# B&R Automation Studio project NAINV104C00R8L515F00 (part 14)

#### Act_OptP1023USSel.st
```iecst
ACTION Act_OptP1023USSel:

	IF tyP1023McSetHComm.tyUSSel.tyBtnSMEMA.bRtCompl = TRUE THEN
		tyP1023McSetHComm.tyUSSel.tyBtnSMEMA.bRtCompl	:= FALSE;

		tyP1023McSetHComm.tyUSSel.tyBtnSMEMA.bValue		:= TRUE;
		tyP1023McSetHComm.tyUSSel.tyBtnSMEMA.bRtLk		:= TRUE;

		tyP1023McSetHComm.tyUSSel.tyBtnHermes.bValue	:= FALSE;
		tyP1023McSetHComm.tyUSSel.tyBtnHermes.bRtLk		:= FALSE;

	ELSIF tyP1023McSetHComm.tyUSSel2.tyBtnSMEMA.bRtCompl = TRUE THEN
		tyP1023McSetHComm.tyUSSel2.tyBtnSMEMA.bRtCompl	:= FALSE;

		tyP1023McSetHComm.tyUSSel2.tyBtnSMEMA.bValue	:= TRUE;
		tyP1023McSetHComm.tyUSSel2.tyBtnSMEMA.bRtLk		:= TRUE;

		tyP1023McSetHComm.tyUSSel2.tyBtnHermes.bValue	:= FALSE;
		tyP1023McSetHComm.tyUSSel2.tyBtnHermes.bRtLk	:= FALSE;

	ELSIF tyP1023McSetHComm.tyUSSel.tyBtnHermes.bRtCompl = TRUE THEN
		tyP1023McSetHComm.tyUSSel.tyBtnHermes.bRtCompl	:= FALSE;

		tyP1023McSetHComm.tyUSSel.tyBtnSMEMA.bValue		:= FALSE;
		tyP1023McSetHComm.tyUSSel.tyBtnSMEMA.bRtLk		:= FALSE;

		tyP1023McSetHComm.tyUSSel.tyBtnHermes.bValue	:= TRUE;
		tyP1023McSetHComm.tyUSSel.tyBtnHermes.bRtLk		:= TRUE;

	ELSIF tyP1023McSetHComm.tyUSSel2.tyBtnHermes.bRtCompl = TRUE THEN //Added
		tyP1023McSetHComm.tyUSSel2.tyBtnHermes.bRtCompl	:= FALSE;

		tyP1023McSetHComm.tyUSSel2.tyBtnSMEMA.bValue	:= FALSE;
		tyP1023McSetHComm.tyUSSel2.tyBtnSMEMA.bRtLk		:= FALSE;

		tyP1023McSetHComm.tyUSSel2.tyBtnHermes.bValue	:= TRUE;
		tyP1023McSetHComm.tyUSSel2.tyBtnHermes.bRtLk	:= TRUE;

	END_IF

	//Upstream Selection

	IF tyP1023McSetHComm.tyGen.tyDrpDnUSSel.bRtCompl THEN

		tyP1023McSetHComm.tyGen.tyDrpDnUSSel.bRtCompl:= FALSE;

		IF tyP1023McSetHComm.tyGen.tyDrpDnUSSel.usiValueIdx = 0 THEN

			p_tyP1023McSetHCommUSSel ACCESS ADR(tyP1023McSetHComm.tyUSSel);
			p_tyP1023McSetHCommUSSMEMA ACCESS ADR(tyP1023McSetHComm.tyUSSMEMA);
			p_tyP1023McSetHCommUSHermes ACCESS ADR(tyP1023McSetHComm.tyUSHermes);

			fUIInRtStatOff(ADR(tyP1023McSetHComm.tyUSSel.tyLyr.uiRtStat));
			fUIInRtStatHide(ADR(tyP1023McSetHComm.tyUSSel2.tyLyr.uiRtStat));

		ELSIF tyP1023McSetHComm.tyGen.tyDrpDnUSSel.usiValueIdx = 1 THEN

			p_tyP1023McSetHCommUSSel ACCESS ADR(tyP1023McSetHComm.tyUSSel2);
			p_tyP1023McSetHCommUSSMEMA ACCESS ADR(tyP1023McSetHComm.tyUSSMEMA2);
			p_tyP1023McSetHCommUSHermes ACCESS ADR(tyP1023McSetHComm.tyUSHermes2);

			fUIInRtStatOff(ADR(tyP1023McSetHComm.tyUSSel2.tyLyr.uiRtStat));
			fUIInRtStatHide(ADR(tyP1023McSetHComm.tyUSSel.tyLyr.uiRtStat));

		END_IF

	END_IF

END_ACTION
```

#### Act_OptP1023DSSel.st
```iecst
ACTION Act_OptP1023DSSel:

	IF tyP1023McSetHComm.tyDSSel.tyBtnSMEMA.bRtCompl = TRUE THEN
		tyP1023McSetHComm.tyDSSel.tyBtnSMEMA.bRtCompl	:= FALSE;

		tyP1023McSetHComm.tyDSSel.tyBtnSMEMA.bValue		:= TRUE;
		tyP1023McSetHComm.tyDSSel.tyBtnSMEMA.bRtLk		:= TRUE;

		tyP1023McSetHComm.tyDSSel.tyBtnHermes.bValue	:= FALSE;
		tyP1023McSetHComm.tyDSSel.tyBtnHermes.bRtLk		:= FALSE;

	ELSIF tyP1023McSetHComm.tyDSSel.tyBtnHermes.bRtCompl = TRUE THEN
		tyP1023McSetHComm.tyDSSel.tyBtnHermes.bRtCompl	:= FALSE;

		tyP1023McSetHComm.tyDSSel.tyBtnSMEMA.bValue		:= FALSE;
		tyP1023McSetHComm.tyDSSel.tyBtnSMEMA.bRtLk		:= FALSE;

		tyP1023McSetHComm.tyDSSel.tyBtnHermes.bValue	:= TRUE;
		tyP1023McSetHComm.tyDSSel.tyBtnHermes.bRtLk		:= TRUE;
	ELSIF tyP1023McSetHComm.tyDSSel2.tyBtnSMEMA.bRtCompl = TRUE THEN
		tyP1023McSetHComm.tyDSSel2.tyBtnSMEMA.bRtCompl	:= FALSE;

		tyP1023McSetHComm.tyDSSel2.tyBtnSMEMA.bValue		:= TRUE;
		tyP1023McSetHComm.tyDSSel2.tyBtnSMEMA.bRtLk		:= TRUE;

		tyP1023McSetHComm.tyDSSel2.tyBtnHermes.bValue	:= FALSE;
		tyP1023McSetHComm.tyDSSel2.tyBtnHermes.bRtLk		:= FALSE;

	ELSIF  tyP1023McSetHComm.tyDSSel2.tyBtnHermes.bRtCompl = TRUE THEN
		tyP1023McSetHComm.tyDSSel2.tyBtnHermes.bRtCompl	:= FALSE;

		tyP1023McSetHComm.tyDSSel2.tyBtnSMEMA.bValue		:= FALSE;
		tyP1023McSetHComm.tyDSSel2.tyBtnSMEMA.bRtLk		:= FALSE;

		tyP1023McSetHComm.tyDSSel2.tyBtnHermes.bValue	:= TRUE;
		tyP1023McSetHComm.tyDSSel2.tyBtnHermes.bRtLk		:= TRUE;

	END_IF

	//Dsstream Selection
	IF tyP1023McSetHComm.tyGen.tyDrpDnDSSel.bRtCompl THEN

		tyP1023McSetHComm.tyGen.tyDrpDnDSSel.bRtCompl:= FALSE;

		IF tyP1023McSetHComm.tyGen.tyDrpDnDSSel.usiValueIdx = 0 THEN

			p_tyP1023McSetHCommDSSel ACCESS ADR(tyP1023McSetHComm.tyDSSel);
			p_tyP1023McSetHCommDSSMEMA ACCESS ADR(tyP1023McSetHComm.tyDSSMEMA);
			p_tyP1023McSetHCommDSHermes ACCESS ADR(tyP1023McSetHComm.tyDSHermes);

			fUIInRtStatOff(ADR(tyP1023McSetHComm.tyDSSel.tyLyr.uiRtStat));
			fUIInRtStatHide(ADR(tyP1023McSetHComm.tyDSSel2.tyLyr.uiRtStat));

		ELSIF tyP1023McSetHComm.tyGen.tyDrpDnDSSel.usiValueIdx = 1 THEN

			p_tyP1023McSetHCommDSSel ACCESS ADR(tyP1023McSetHComm.tyDSSel2);
			p_tyP1023McSetHCommDSSMEMA ACCESS ADR(tyP1023McSetHComm.tyDSSMEMA2);
			p_tyP1023McSetHCommDSHermes ACCESS ADR(tyP1023McSetHComm.tyDSHermes2);

			fUIInRtStatOff(ADR(tyP1023McSetHComm.tyDSSel2.tyLyr.uiRtStat));
			fUIInRtStatHide(ADR(tyP1023McSetHComm.tyDSSel.tyLyr.uiRtStat));

		END_IF

	END_IF

END_ACTION
```

#### Act_OptP1023Keypad.st
```iecst
ACTION Act_OptP1023Keypad:

	IF fUIOutRtStatTPIsOpen(ADR(tyP1023McSetHComm.tyUSHermes.tyNumSndAliveTm.uiRtStat)) = TRUE THEN
		tyProperty.tyKeypad.tyTxtTitle.sTxt	:= tyP1023McSetHComm.tyUSHermes.tyNumSndAliveTm.sKeypadTitle;

	ELSIF fUIOutRtStatTPIsOpen(ADR(tyP1023McSetHComm.tyUSHermes.tyNumLaneID.uiRtStat)) = TRUE THEN
		tyProperty.tyKeypad.tyTxtTitle.sTxt	:= tyP1023McSetHComm.tyUSHermes.tyNumLaneID.sKeypadTitle;

	ELSIF fUIOutRtStatTPIsOpen(ADR(tyP1023McSetHComm.tyUSHermes.tyStringHostAddr.uiRtStat)) = TRUE THEN
		tyProperty.tyKeypad.tyTxtTitle.sTxt	:= tyP1023McSetHComm.tyUSHermes.tyStringHostAddr.sKeypadTitle;

	ELSIF fUIOutRtStatTPIsOpen(ADR(tyP1023McSetHComm.tyUSHermes.tyNumHostPort.uiRtStat)) = TRUE THEN
		tyProperty.tyKeypad.tyTxtTitle.sTxt	:= tyP1023McSetHComm.tyUSHermes.tyNumHostPort.sKeypadTitle;

	ELSIF fUIOutRtStatTPIsOpen(ADR(tyP1023McSetHComm.tyDSHermes.tyNumSndAliveTm.uiRtStat)) = TRUE THEN
		tyProperty.tyKeypad.tyTxtTitle.sTxt	:= tyP1023McSetHComm.tyDSHermes.tyNumSndAliveTm.sKeypadTitle;

	ELSIF fUIOutRtStatTPIsOpen(ADR(tyP1023McSetHComm.tyDSHermes.tyNumLaneID.uiRtStat)) = TRUE THEN
		tyProperty.tyKeypad.tyTxtTitle.sTxt	:= tyP1023McSetHComm.tyDSHermes.tyNumLaneID.sKeypadTitle;

	ELSIF fUIOutRtStatTPIsOpen(ADR(tyP1023McSetHComm.tyDSHermes.tyNumSvrPort.uiRtStat)) = TRUE THEN
		tyProperty.tyKeypad.tyTxtTitle.sTxt	:= tyP1023McSetHComm.tyDSHermes.tyNumSvrPort.sKeypadTitle;

	END_IF

END_ACTION
```

#### Act_EntP1024Disp.st
```iecst
ACTION Act_EntP1024Disp:

	//Access Address
	p_tyC0004Navi ACCESS ADR(tyP1024McSetAntiGap.tyNaviBack);

	p_tyC0005Main ACCESS ADR(tyCommon.tyMain);

	p_tyC0006Set ACCESS ADR(tyCommon.tySet);

	p_tyC0007Notif ACCESS ADR(tyCommon.tyNotif);

	p_tyC0008MsgBox ACCESS ADR(tyP1024McSetAntiGap.tyMsgBoxHide);

	p_tyC0009Info ACCESS ADR(tyCommon.tyInfo);

	p_tyC0011Loading ACCESS ADR(tyCommon.tyLoading);

	p_tyP1024McSetAntiGap ACCESS ADR(tyP1024McSetAntiGap.tyAntiGap);

	//Backup Param
	tyP1024McSetAntiGap.tyAntiGapBkUp	:= tyP1024McSetAntiGap.tyAntiGap;

END_ACTION
```

#### Act_ExitP1024.st
```iecst
ACTION Act_ExitP1024:

	IF tyCommon.tySet.tyBtnSave.uiMaskRtStat.0 = FALSE THEN
		usiChgPage	:= 1;

	ELSE

		p_tyC0008MsgBox ACCESS ADR(tyP1024McSetAntiGap.tyMsgBoxExitAsk);

		IF tyP1024McSetAntiGap.tyMsgBoxExitAsk.tyBtnYes.bRtCompl = TRUE THEN
			tyP1024McSetAntiGap.tyMsgBoxExitAsk.tyBtnYes.bRtCompl	:= FALSE;
			tyP1024McSetAntiGap.tyMsgBoxExitAsk.tyBtnYes.bValue		:= FALSE;

			p_tyC0008MsgBox ACCESS ADR(tyP1024McSetAntiGap.tyMsgBoxHide);

			//Restore Param
			tyP1024McSetAntiGap.tyAntiGap	:= tyP1024McSetAntiGap.tyAntiGapBkUp;

			fUIInRtStatOff(ADR(tyCommon.tySet.tyBtnSave.uiMaskRtStat));

			usiChgPage	:= 1;

		ELSIF tyP1024McSetAntiGap.tyMsgBoxExitAsk.tyBtnNo.bRtCompl = TRUE THEN
			tyP1024McSetAntiGap.tyMsgBoxExitAsk.tyBtnNo.bRtCompl	:= FALSE;
			tyP1024McSetAntiGap.tyMsgBoxExitAsk.tyBtnNo.bValue		:= FALSE;

			p_tyC0008MsgBox ACCESS ADR(tyP1024McSetAntiGap.tyMsgBoxHide);

			eChgPage	:= eCurrPage;
			usiChgPage	:= 0;

		END_IF

	END_IF

END_ACTION
```

#### Act_OptP1024Navi.st
```iecst
ACTION Act_OptP1024Navi:

	IF tyP1024McSetAntiGap.tyNaviBack.tyBtnBack.bRtCompl = TRUE THEN
		tyP1024McSetAntiGap.tyNaviBack.tyBtnBack.bRtCompl	:= FALSE;

		eChgPage	:= UIP1020McSetNavi;

	END_IF

END_ACTION
```

#### Act_OptP1024Save.st
```iecst
ACTION Act_OptP1024Save:

	IF 	tyP1024McSetAntiGap.tyAntiGap.tyNumLftSenOff.bRtCompl OR tyP1024McSetAntiGap.tyAntiGap.tyNumRgtSenOff.bRtCompl THEN

		fUIInRtStatHide(ADR(tyCommon.tySet.tyBtnSave.uiMaskRtStat));

		tyP1024McSetAntiGap.tyAntiGap.tyNumLftSenOff.bRtCompl	:= FALSE;
		tyP1024McSetAntiGap.tyAntiGap.tyNumRgtSenOff.bRtCompl	:= FALSE;

	END_IF

	IF tyCommon.tySet.tyBtnSave.bRtCompl = TRUE THEN
		//Save Param
		tyMcParamWr.tyConvLftSenAntiGapDly.diSigOffTm	:= tyP1024McSetAntiGap.tyAntiGap.tyNumLftSenOff.diValue;
		tyMcParamWr.tyConvRgtSenAntiGapDly.diSigOffTm	:= tyP1024McSetAntiGap.tyAntiGap.tyNumRgtSenOff.diValue;

		eMcParamAct	:= McParamActWrite;

		IF p_eMcParamStat = McParamActWrite AND p_eMcParamStatus = Done THEN
			eMcParamAct	:= McParamActIdle;

			//Backup Param
			tyP1024McSetAntiGap.tyAntiGapBkUp	:= tyP1024McSetAntiGap.tyAntiGap;

			tyCommon.tySet.tyBtnSave.bRtCompl	:= FALSE;

			fUIInRtStatOff(ADR(tyCommon.tySet.tyBtnSave.uiMaskRtStat));

		ELSIF p_eMcParamStatus = Error THEN
			p_tyC0008MsgBox ACCESS ADR(tyP1024McSetAntiGap.tyMsgBoxSaveErr);

			IF tyP1021McSetGen.tyMsgBoxSaveErr.tyBtnNo.bRtCompl = TRUE THEN
				tyP1021McSetGen.tyMsgBoxSaveErr.tyBtnNo.bRtCompl	:= FALSE;
				tyP1021McSetGen.tyMsgBoxSaveErr.tyBtnNo.bValue		:= FALSE;

				p_tyC0008MsgBox ACCESS ADR(tyP1024McSetAntiGap.tyMsgBoxHide);

				//Restore Param
				tyP1024McSetAntiGap.tyAntiGap	:= tyP1024McSetAntiGap.tyAntiGapBkUp;
				tyMcParamWr						:= p_tyMcParamCurr;

				tyCommon.tySet.tyBtnSave.bRtCompl	:= FALSE;

				fUIInRtStatOff(ADR(tyCommon.tySet.tyBtnSave.uiMaskRtStat));

			END_IF

		END_IF

	END_IF

END_ACTION
```

#### Act_OptP1024Keypad.st
```iecst
ACTION Act_OptP1024Keypad:

	IF fUIOutRtStatTPIsOpen(ADR(tyP1024McSetAntiGap.tyAntiGap.tyNumLftSenOff.uiRtStat)) = TRUE THEN
		tyProperty.tyKeypad.tyTxtTitle.sTxt	:= tyP1024McSetAntiGap.tyAntiGap.tyNumLftSenOff.sKeypadTitle;

	ELSIF fUIOutRtStatTPIsOpen(ADR(tyP1024McSetAntiGap.tyAntiGap.tyNumRgtSenOff.uiRtStat)) = TRUE THEN
		tyProperty.tyKeypad.tyTxtTitle.sTxt	:= tyP1024McSetAntiGap.tyAntiGap.tyNumRgtSenOff.sKeypadTitle;

	END_IF

END_ACTION
```

#### Act_EntP1040Disp.st
```iecst
ACTION Act_EntP1040Disp:

	//Access Address
	p_tyC0005Main ACCESS ADR(tyCommon.tyMain);

	p_tyC0007Notif ACCESS ADR(tyCommon.tyNotif);

	p_tyC0008MsgBox ACCESS ADR(tyP1040ProdSet.tyMsgBoxHide);

	p_tyC0009Info ACCESS ADR(tyCommon.tyInfo);

	p_tyC0011Loading ACCESS ADR(tyCommon.tyLoading);

	p_tyC0012RcpPopUp ACCESS ADR(tyP1040ProdSet.tyRcpPopUp);

	p_tyP1040ProdSet ACCESS ADR(tyP1040ProdSet.tyProdSet);

	//Display
	tyP1040ProdSet.tyProdSet.tyStringSearch.sValue	:= '';
	udiP1040SelectedRowOld	 := 0;

	fUIInRtStatHide(ADR(tyP1040ProdSet.tyRcpPopUp.tyLyr.uiRtStat));

	tyP1040ProdSet.tyProdSet.tyBtnSort.bValue := FALSE;
	tyP1040ProdSet.tyProdSet.tyBtnSort.bRtCompl := FALSE;

END_ACTION
```

#### Act_OptP1040Mask.st
```iecst
ACTION Act_OptP1040Mask:

	IF tyP1040ProdSet.tyProdSet.tyNumProdWidth.bRtCompl 			OR tyP1040ProdSet.tyProdSet.tyStringRecipeNm.bRtCompl
		OR tyP1040ProdSet.tyProdSet.tyDrpDnMcMode.bRtCompl 			OR tyP1040ProdSet.tyProdSet.tyDrpDnFlippedBrd.bRtCompl
		OR tyP1040ProdSet.tyProdSet.tyStringMatchCode.bRtCompl 		OR tyP1040ProdSet.tyProdSet.tyNumProdWidth2.bRtCompl THEN

		fUIInRtStatHide(ADR(tyP1040ProdSet.tyProdSet.tyBtnSave.uiMaskRtStat));

		tyP1040ProdSet.tyProdSet.tyStringRecipeNm.bRtCompl	:= FALSE;
		tyP1040ProdSet.tyProdSet.tyNumProdWidth.bRtCompl	:= FALSE;
		tyP1040ProdSet.tyProdSet.tyNumProdWidth2.bRtCompl	:= FALSE;
		tyP1040ProdSet.tyProdSet.tyDrpDnMcMode.bRtCompl		:= FALSE;
		tyP1040ProdSet.tyProdSet.tyDrpDnFlippedBrd.bRtCompl	:= FALSE;
		tyP1040ProdSet.tyProdSet.tyStringMatchCode.bRtCompl	:= FALSE;
	END_IF

	IF (tyP1040ProdSet.tyProdSet.tyTableRecipe.a_tyStringDataCol1[tyP1040Table.uiSelectedRow].sValue <> '') AND (tyP1040ProdSet.tyProdSet.tyBtnSave.bRtCompl = FALSE) AND (tyP1040ProdSet.tyProdSet.tyBtnToXML.bRtCompl = FALSE) AND (tyP1040ProdSet.tyProdSet.tyBtnFromXML.bRtCompl = FALSE) THEN
		fUIInRtStatHide(ADR(tyP1040ProdSet.tyProdSet.tyBtnDelete.uiMaskRtStat));
	ELSE
		fUIInRtStatOff(ADR(tyP1040ProdSet.tyProdSet.tyBtnDelete.uiMaskRtStat));
	END_IF

	tyP1040ProdSet.tyProdSet.tyBtnToXML.uiMaskRtStat.0		:= (tyP1040ProdSet.tyProdSet.tyBtnSave.uiMaskRtStat.0 = FALSE) AND (tyP1040ProdSet.tyProdSet.tyBtnDelete.bRtCompl = FALSE) AND (tyP1040ProdSet.tyProdSet.tyBtnFromXML.bRtCompl = FALSE);
	tyP1040ProdSet.tyProdSet.tyBtnFromXML.uiMaskRtStat.0	:= (tyP1040ProdSet.tyProdSet.tyBtnSave.uiMaskRtStat.0 = FALSE) AND (tyP1040ProdSet.tyProdSet.tyBtnDelete.bRtCompl = FALSE) AND (tyP1040ProdSet.tyProdSet.tyBtnToXML.bRtCompl = FALSE);

	tyP1040ProdSet.tyProdSet.tyBtnSort.uiMaskRtStat.0		:= (tyP1040ProdSet.tyProdSet.tyTableRecipe.a_tyStringDataCol1[1].sValue <> '') AND (tyP1040ProdSet.tyProdSet.tyStringSearch.bRtCompl = FALSE)
																AND (tyP1040ProdSet.tyProdSet.tyBtnSave.uiMaskRtStat.0 = FALSE) AND (tyP1040ProdSet.tyProdSet.tyBtnDelete.bRtCompl = FALSE)
																AND (tyP1040ProdSet.tyProdSet.tyBtnToXML.bRtCompl = FALSE) AND (tyP1040ProdSet.tyProdSet.tyBtnFromXML.bRtCompl = FALSE);

END_ACTION
```

#### Act_OptP1040Save.st
```iecst
ACTION Act_OptP1040Save:

	IF tyP1040ProdSet.tyProdSet.tyBtnSave.bRtCompl = TRUE THEN

		IF usiSaveProdRcpStep = 0 THEN
			//Mask
			tyP1040ProdSet.tyProdSet.tyStringSearch.uiMaskRtStat	:= FALSE;
			tyP1040ProdSet.tyProdSet.tyTableRecipe.uiMaskRtStat		:= FALSE;
			tyP1040ProdSet.tyProdSet.tyBtnDelete.uiMaskRtStat					:= FALSE;

			p_tyC0008MsgBox ACCESS ADR(tyP1040ProdSet.tyMsgBoxSaveAsk);

			IF tyP1040ProdSet.tyMsgBoxSaveAsk.tyBtnYes.bRtCompl = TRUE THEN
				tyP1040ProdSet.tyMsgBoxSaveAsk.tyBtnYes.bRtCompl	:= FALSE;
				tyP1040ProdSet.tyMsgBoxSaveAsk.tyBtnYes.bValue		:= FALSE;

				p_tyC0008MsgBox ACCESS ADR(tyP1040ProdSet.tyMsgBoxHide);

				usiSaveProdRcpStep	:= 1;

			ELSIF tyP1040ProdSet.tyMsgBoxSaveAsk.tyBtnNo.bRtCompl = TRUE THEN
				tyP1040ProdSet.tyMsgBoxSaveAsk.tyBtnNo.bRtCompl	:= FALSE;
				tyP1040ProdSet.tyMsgBoxSaveAsk.tyBtnNo.bValue	:= FALSE;

				p_tyC0008MsgBox ACCESS ADR(tyP1040ProdSet.tyMsgBoxHide);

				usiSaveProdRcpStep	:= 99;

			END_IF

		ELSIF usiSaveProdRcpStep = 1 THEN
			tyProdRcpInfoIn.sRcpNm			:= tyP1040ProdSet.tyProdSet.tyStringRecipeNm.sValue;
			tyProdRcpInfoIn.diWidthInUM		:= tyP1040ProdSet.tyProdSet.tyNumProdWidth.diValue;
			tyProdRcpInfoIn.usiMcMod		:= tyP1040ProdSet.tyProdSet.tyDrpDnMcMode.usiValueIdx;
			tyProdRcpInfoIn.usiFlippedBrd	:= tyP1040ProdSet.tyProdSet.tyDrpDnFlippedBrd.usiValueIdx;
			tyProdRcpInfoIn.sMatchCode		:= tyP1040ProdSet.tyProdSet.tyStringMatchCode.sValue;

			IF p_tyNtParamCurr.bLFProdWidth2Prep THEN
				tyProdRcpInfoIn.diWidthInUM2		:= tyP1040ProdSet.tyProdSet.tyNumProdWidth2.diValue;// ADD
			ELSE
				tyProdRcpInfoIn.diWidthInUM2		:= tyP1040ProdSet.tyProdSet.tyNumProdWidth.diValue;// ADD
			END_IF

			eProdRcpAct	:= ProdRcpActAddEdit;

			IF p_eProdRcpStat = ProdRcpActAddEdit AND p_eProdRcpStatus = Done THEN
				eProdRcpAct	:= ProdRcpActIdle;

				IF p_bProdRcpNmEmpty = TRUE THEN
					usiSaveProdRcpStep		:= 2;
				ELSIF p_bProdRcpListFull = TRUE THEN
					usiSaveProdRcpStep		:= 3;
				ELSE
					fUIInRtStatOff(ADR(tyP1040ProdSet.tyProdSet.tyBtnSave.uiMaskRtStat));
					tyP1040ProdSet.tyProdSet.tyBtnSort.bValue := FALSE;
					tyP1040ProdSet.tyProdSet.tyStringSearch.sValue := '';

					bRefreshProdRcpTable	:= TRUE;
					bRefreshProdRcpDetail	:= TRUE;
					usiSaveProdRcpStep		:= 4;
				END_IF

			ELSIF p_eProdRcpStatus = Error THEN
				p_tyC0008MsgBox ACCESS ADR(tyP1040ProdSet.tyMsgBoxSaveErr);

				IF tyP1040ProdSet.tyMsgBoxSaveErr.tyBtnNo.bRtCompl = TRUE THEN
					tyP1040ProdSet.tyMsgBoxSaveErr.tyBtnNo.bRtCompl	:= FALSE;
					tyP1040ProdSet.tyMsgBoxSaveErr.tyBtnNo.bValue 	:= FALSE;

					p_tyC0008MsgBox ACCESS ADR(tyP1040ProdSet.tyMsgBoxHide);

					usiSaveProdRcpStep	:= 99;
				END_IF

			END_IF

			//Product Recipe Parameter Error
		ELSIF usiSaveProdRcpStep = 2 THEN
			p_tyC0008MsgBox ACCESS ADR(tyP1040ProdSet.tyMsgBoxSaveNoNm);

			IF tyP1040ProdSet.tyMsgBoxSaveNoNm.tyBtnNo.bRtCompl = TRUE THEN
				tyP1040ProdSet.tyMsgBoxSaveNoNm.tyBtnNo.bRtCompl	:= FALSE;
				tyP1040ProdSet.tyMsgBoxSaveNoNm.tyBtnNo.bValue 		:= FALSE;

				p_tyC0008MsgBox ACCESS ADR(tyP1040ProdSet.tyMsgBoxHide);

				usiSaveProdRcpStep	:= 99;
			END_IF

			//Product Recipe List Full
		ELSIF usiSaveProdRcpStep = 3 THEN
			p_tyC0008MsgBox ACCESS ADR(tyP1040ProdSet.tyMsgBoxListFull);

			IF tyP1040ProdSet.tyMsgBoxListFull.tyBtnNo.bRtCompl = TRUE THEN
				tyP1040ProdSet.tyMsgBoxListFull.tyBtnNo.bRtCompl	:= FALSE;
				tyP1040ProdSet.tyMsgBoxListFull.tyBtnNo.bValue 		:= FALSE;

				p_tyC0008MsgBox ACCESS ADR(tyP1040ProdSet.tyMsgBoxHide);

				usiSaveProdRcpStep	:= 99;
			END_IF

		ELSIF usiSaveProdRcpStep = 4 THEN
			IF tyProdRcpInfoIn.sRcpNm = p_tyProdRcpCurrRcp0.sRcpNm THEN
				p_tyC0008MsgBox ACCESS ADR(tyP1040ProdSet.tyMsgBoxReloadCurrRcp);

				IF tyP1040ProdSet.tyMsgBoxReloadCurrRcp.tyBtnNo.bRtCompl = TRUE THEN
					tyP1040ProdSet.tyMsgBoxReloadCurrRcp.tyBtnNo.bRtCompl	:= FALSE;
					tyP1040ProdSet.tyMsgBoxReloadCurrRcp.tyBtnNo.bValue 	:= FALSE;

					p_tyC0008MsgBox ACCESS ADR(tyP1040ProdSet.tyMsgBoxHide);

					usiSaveProdRcpStep	:= 99;
				END_IF
			ELSE
				usiSaveProdRcpStep	:= 99;
			END_IF

		ELSIF usiSaveProdRcpStep = 99 THEN
			bRefreshProdRcpTable	:= FALSE;

			//Unmask
			tyP1040ProdSet.tyProdSet.tyStringSearch.uiMaskRtStat	:= TRUE;
			tyP1040ProdSet.tyProdSet.tyTableRecipe.uiMaskRtStat		:= TRUE;
			tyP1040ProdSet.tyProdSet.tyBtnDelete.uiMaskRtStat		:= TRUE;

			//Reset
			tyP1040ProdSet.tyProdSet.tyBtnSave.bRtCompl	:= FALSE;
			tyP1040ProdSet.tyProdSet.tyBtnSave.bValue	:= FALSE;

			usiSaveProdRcpStep	:= 0;

		END_IF

	END_IF

END_ACTION
```

#### Act_OptP1040LoadData.st
```iecst
ACTION Act_OptP1040LoadData:

	udiP1040SelectedRow	:= STRING_TO_UDINT(tyP1040ProdSet.tyProdSet.tyTableRecipe.a_tyStringDataCol0[tyP1040Table.uiSelectedRow].sValue);

	IF udiP1040SelectedRow <> udiP1040SelectedRowOld OR bRefreshProdRcpDetail = TRUE OR bUpdateP1040LoadData OR bUpdateP1040LoadData THEN

		IF tyP1040ProdSet.tyProdSet.tyStringSearch.sValue = '' THEN

			IF tyP1040ProdSet.tyProdSet.tyTableRecipe.a_tyStringDataCol1[tyP1040Table.uiSelectedRow].sValue <> '' THEN
				//Update Recipe Data
				IF tyP1040ProdSet.tyProdSet.tyBtnSort.bValue THEN
					tyP1040ProdSet.tyProdSet.tyStringRecipeNm.sValue				:= p_tyProdRcpSortedList[udiP1040SelectedRow].sRcpNm;
					tyP1040ProdSet.tyProdSet.tyNumProdWidth.diValue					:= p_tyProdRcpSortedList[udiP1040SelectedRow].diWidthInUM;
					tyP1040ProdSet.tyProdSet.tyNumProdWidth2.diValue				:= p_tyProdRcpSortedList[udiP1040SelectedRow].diWidthInUM2;
					tyP1040ProdSet.tyProdSet.tyDrpDnMcMode.usiValueIdx				:= p_tyProdRcpSortedList[udiP1040SelectedRow].usiMcMod;
					tyP1040ProdSet.tyProdSet.tyDrpDnFlippedBrd.usiValueIdx			:= p_tyProdRcpSortedList[udiP1040SelectedRow].usiFlippedBrd;
					tyP1040ProdSet.tyProdSet.tyStringMatchCode.sValue				:= p_tyProdRcpSortedList[udiP1040SelectedRow].sMatchCode;
				ELSE
					tyP1040ProdSet.tyProdSet.tyStringRecipeNm.sValue				:= p_tyProdRcpCurrList[udiP1040SelectedRow].sRcpNm;
					tyP1040ProdSet.tyProdSet.tyNumProdWidth.diValue					:= p_tyProdRcpCurrList[udiP1040SelectedRow].diWidthInUM;
					tyP1040ProdSet.tyProdSet.tyNumProdWidth2.diValue				:= p_tyProdRcpCurrList[udiP1040SelectedRow].diWidthInUM2;
					tyP1040ProdSet.tyProdSet.tyDrpDnMcMode.usiValueIdx				:= p_tyProdRcpCurrList[udiP1040SelectedRow].usiMcMod;
					tyP1040ProdSet.tyProdSet.tyDrpDnFlippedBrd.usiValueIdx			:= p_tyProdRcpCurrList[udiP1040SelectedRow].usiFlippedBrd;
					tyP1040ProdSet.tyProdSet.tyStringMatchCode.sValue				:= p_tyProdRcpCurrList[udiP1040SelectedRow].sMatchCode;
				END_IF
			ELSE
				//Defaut Recipe Data
				tyP1040ProdSet.tyProdSet.tyStringRecipeNm.sValue				:= '';
				tyP1040ProdSet.tyProdSet.tyNumProdWidth.diValue					:= 100000;
				tyP1040ProdSet.tyProdSet.tyNumProdWidth2.diValue				:= 100000;
				tyP1040ProdSet.tyProdSet.tyDrpDnMcMode.usiValueIdx				:= p_tyMcParamCurr.usiDefaultMcMod;
				tyP1040ProdSet.tyProdSet.tyDrpDnFlippedBrd.usiValueIdx			:= p_tyMcParamCurr.usiDefaultFlippedBrd;
				tyP1040ProdSet.tyProdSet.tyStringMatchCode.sValue				:= '';
			END_IF

		ELSE

			IF tyP1040ProdSet.tyProdSet.tyTableRecipe.a_tyStringDataCol1[tyP1040Table.uiSelectedRow].sValue <> '' THEN
				//Update Recipe Data
				IF tyP1040ProdSet.tyProdSet.tyBtnSort.bValue THEN
					tyP1040ProdSet.tyProdSet.tyStringRecipeNm.sValue				:= p_tyProdRcpSortedList[udiP1040SelectedRow].sRcpNm;
					tyP1040ProdSet.tyProdSet.tyNumProdWidth.diValue					:= p_tyProdRcpSortedList[udiP1040SelectedRow].diWidthInUM;
					tyP1040ProdSet.tyProdSet.tyNumProdWidth2.diValue				:= p_tyProdRcpSortedList[udiP1040SelectedRow].diWidthInUM2;
					tyP1040ProdSet.tyProdSet.tyDrpDnMcMode.usiValueIdx				:= p_tyProdRcpSortedList[udiP1040SelectedRow].usiMcMod;
					tyP1040ProdSet.tyProdSet.tyDrpDnFlippedBrd.usiValueIdx			:= p_tyProdRcpSortedList[udiP1040SelectedRow].usiFlippedBrd;
					tyP1040ProdSet.tyProdSet.tyStringMatchCode.sValue				:= p_tyProdRcpSortedList[udiP1040SelectedRow].sMatchCode;

				ELSE
					tyP1040ProdSet.tyProdSet.tyStringRecipeNm.sValue				:= p_tyProdRcpFilterList[udiP1040SelectedRow].sRcpNm;
					tyP1040ProdSet.tyProdSet.tyNumProdWidth.diValue					:= p_tyProdRcpFilterList[udiP1040SelectedRow].diWidthInUM;
					tyP1040ProdSet.tyProdSet.tyNumProdWidth2.diValue				:= p_tyProdRcpFilterList[udiP1040SelectedRow].diWidthInUM2;
					tyP1040ProdSet.tyProdSet.tyDrpDnMcMode.usiValueIdx				:= p_tyProdRcpFilterList[udiP1040SelectedRow].usiMcMod;
					tyP1040ProdSet.tyProdSet.tyDrpDnFlippedBrd.usiValueIdx			:= p_tyProdRcpFilterList[udiP1040SelectedRow].usiFlippedBrd;
					tyP1040ProdSet.tyProdSet.tyStringMatchCode.sValue				:= p_tyProdRcpFilterList[udiP1040SelectedRow].sMatchCode;
				END_IF

			ELSE
				//Defaut Recipe Data
				tyP1040ProdSet.tyProdSet.tyStringRecipeNm.sValue				:= '';
				tyP1040ProdSet.tyProdSet.tyNumProdWidth.diValue					:= 100000;
				tyP1040ProdSet.tyProdSet.tyNumProdWidth2.diValue				:= 100000;
				tyP1040ProdSet.tyProdSet.tyDrpDnMcMode.usiValueIdx				:= p_tyMcParamCurr.usiDefaultMcMod;
				tyP1040ProdSet.tyProdSet.tyDrpDnFlippedBrd.usiValueIdx			:= p_tyMcParamCurr.usiDefaultFlippedBrd;
				tyP1040ProdSet.tyProdSet.tyStringMatchCode.sValue				:= '';
			END_IF

		END_IF

		bUpdateP1040LoadData	:= FALSE;
		bRefreshProdRcpDetail	:= FALSE;
		udiP1040SelectedRowOld	:= udiP1040SelectedRow;

		fUIInRtStatOff(ADR(tyP1040ProdSet.tyProdSet.tyBtnSave.uiMaskRtStat));

	END_IF

END_ACTION
```

#### Act_OptP1040Del.st
```iecst
ACTION Act_OptP1040Del:

	IF tyP1040ProdSet.tyProdSet.tyBtnDelete.bRtCompl = TRUE THEN

		IF usiDelProdRcpStep = 0 THEN
			//Mask
			tyP1040ProdSet.tyProdSet.tyStringSearch.uiMaskRtStat	:= FALSE;
			tyP1040ProdSet.tyProdSet.tyTableRecipe.uiMaskRtStat		:= FALSE;

			IF tyP1040ProdSet.tyProdSet.tyTableRecipe.a_tyStringDataCol1[tyP1040Table.uiSelectedRow].sValue = p_tyProdRcpCurrRcp0.sRcpNm THEN
				p_tyC0008MsgBox ACCESS ADR(tyP1040ProdSet.tyMsgBoxDelCurrRcpAsk);

				IF tyP1040ProdSet.tyMsgBoxDelCurrRcpAsk.tyBtnNo.bRtCompl = TRUE THEN
					tyP1040ProdSet.tyMsgBoxDelCurrRcpAsk.tyBtnNo.bRtCompl	:= FALSE;
					tyP1040ProdSet.tyMsgBoxDelCurrRcpAsk.tyBtnNo.bValue		:= FALSE;

					p_tyC0008MsgBox ACCESS ADR(tyP1040ProdSet.tyMsgBoxHide);

					usiDelProdRcpStep	:= 99;
				END_IF

			ELSE

				p_tyC0008MsgBox ACCESS ADR(tyP1040ProdSet.tyMsgBoxDelAsk);

				IF tyP1040ProdSet.tyMsgBoxDelAsk.tyBtnYes.bRtCompl = TRUE THEN
					tyP1040ProdSet.tyMsgBoxDelAsk.tyBtnYes.bRtCompl	:= FALSE;
					tyP1040ProdSet.tyMsgBoxDelAsk.tyBtnYes.bValue	:= FALSE;

					p_tyC0008MsgBox ACCESS ADR(tyP1040ProdSet.tyMsgBoxHide);

					usiDelProdRcpStep	:= 1;

				ELSIF tyP1040ProdSet.tyMsgBoxDelAsk.tyBtnNo.bRtCompl = TRUE THEN
					tyP1040ProdSet.tyMsgBoxDelAsk.tyBtnNo.bRtCompl	:= FALSE;
					tyP1040ProdSet.tyMsgBoxDelAsk.tyBtnNo.bValue	:= FALSE;

					p_tyC0008MsgBox ACCESS ADR(tyP1040ProdSet.tyMsgBoxHide);

					usiDelProdRcpStep	:= 99;
				END_IF

			END_IF

		ELSIF usiDelProdRcpStep = 1 THEN
			tyProdRcpInfoIn.sRcpNm	:= tyP1040ProdSet.tyProdSet.tyTableRecipe.a_tyStringDataCol1[tyP1040Table.uiSelectedRow].sValue;

			eProdRcpAct	:= ProdRcpActDel;

			IF p_eProdRcpStat = ProdRcpActDel AND p_eProdRcpStatus = Done THEN
				eProdRcpAct	:= ProdRcpActIdle;

				IF p_bProdRcpNmEmpty = TRUE THEN
					usiDelProdRcpStep		:= 2;
				ELSIF p_bProdRcpNmNotExist = TRUE THEN
					usiDelProdRcpStep		:= 3;
				ELSE
					tyP1040ProdSet.tyProdSet.tyBtnSort.bValue := FALSE;
					tyP1040ProdSet.tyProdSet.tyStringSearch.sValue := '';

					bRefreshProdRcpTable	:= TRUE;
					bRefreshProdRcpDetail	:= TRUE;
					usiDelProdRcpStep		:= 99;
				END_IF

			ELSIF p_eProdRcpStatus = Error THEN
				p_tyC0008MsgBox ACCESS ADR(tyP1040ProdSet.tyMsgBoxDelErr);

				IF tyP1040ProdSet.tyMsgBoxDelErr.tyBtnNo.bRtCompl = TRUE THEN
					tyP1040ProdSet.tyMsgBoxDelErr.tyBtnNo.bRtCompl	:= FALSE;
					tyP1040ProdSet.tyMsgBoxDelErr.tyBtnNo.bValue	:= FALSE;

					p_tyC0008MsgBox ACCESS ADR(tyP1040ProdSet.tyMsgBoxHide);

					usiDelProdRcpStep	:= 99;
				END_IF

			END_IF

		ELSIF usiDelProdRcpStep = 2 THEN
			p_tyC0008MsgBox ACCESS ADR(tyP1040ProdSet.tyMsgBoxDelNmEmpty);

			IF tyP1040ProdSet.tyMsgBoxDelNmEmpty.tyBtnNo.bRtCompl = TRUE THEN
				tyP1040ProdSet.tyMsgBoxDelNmEmpty.tyBtnNo.bRtCompl	:= FALSE;
				tyP1040ProdSet.tyMsgBoxDelNmEmpty.tyBtnNo.bValue	:= FALSE;

				p_tyC0008MsgBox ACCESS ADR(tyP1040ProdSet.tyMsgBoxHide);

				usiDelProdRcpStep	:= 99;
			END_IF

		ELSIF usiDelProdRcpStep = 3 THEN
			p_tyC0008MsgBox ACCESS ADR(tyP1040ProdSet.tyMsgBoxDelNmNotExist);

			IF tyP1040ProdSet.tyMsgBoxDelNmNotExist.tyBtnNo.bRtCompl = TRUE THEN
				tyP1040ProdSet.tyMsgBoxDelNmNotExist.tyBtnNo.bRtCompl	:= FALSE;
				tyP1040ProdSet.tyMsgBoxDelNmNotExist.tyBtnNo.bValue		:= FALSE;

				p_tyC0008MsgBox ACCESS ADR(tyP1040ProdSet.tyMsgBoxHide);

				usiDelProdRcpStep	:= 99;
			END_IF

		ELSIF usiDelProdRcpStep = 99 THEN
			bRefreshProdRcpTable	:= FALSE;

			//Unmask
			tyP1040ProdSet.tyProdSet.tyStringSearch.uiMaskRtStat	:= TRUE;
			tyP1040ProdSet.tyProdSet.tyTableRecipe.uiMaskRtStat		:= TRUE;

			//Reset
			tyP1040ProdSet.tyProdSet.tyBtnDelete.bRtCompl	:= FALSE;
			tyP1040ProdSet.tyProdSet.tyBtnDelete.bValue		:= FALSE;

			usiDelProdRcpStep	:= 0;

		END_IF

	END_IF

END_ACTION
```

#### Act_OptP1040Table.st
```iecst
ACTION Act_OptP1040Table:

	//Call Table FB
	fbP1040Table.sVisuNm			:= tyP1040Table.sVisuNm;
	fbP1040Table.udiWorkAreaStartX	:= 359;
	fbP1040Table.udiWorkAreaEndX	:= 770;
	fbP1040Table.udiWorkAreaStartY	:= 93;
	fbP1040Table.udiWorkAreaEndY	:= 415;
	fbP1040Table.udiMinXDist		:= 20;
	fbP1040Table.udiMinYDist		:= 20;
	fbP1040Table.uiSlideScale		:= c_uiP1040TableSize;
	fbP1040Table.iTotalData			:= UDINT_TO_INT(c_udiProdRcpMax);
	fbP1040Table.iTotalRow			:= c_uiP1040TableSize;
	fbP1040Table.p_uiSliderStatus	:= ADR(tyP1040ProdSet.tyProdSet.tyTableRecipe.tyUISlider.uiRtStat);
	fbP1040Table.pa_tyUIHotspot		:= ADR(tyP1040ProdSet.tyProdSet.tyTableRecipe.a_tyHotspot);
	fbP1040Table.p_uiTablePos		:= ADR(tyP1040Table.uiTablePos);
	fbP1040Table.p_iSliderPos		:= ADR(tyP1040ProdSet.tyProdSet.tyTableRecipe.tyUISlider.iValue);
	fbP1040Table.p_uiSelectedRow	:= ADR(tyP1040Table.uiSelectedRow);
	fbP1040Table.p_bTableActive		:= ADR(tyP1040Table.bTableActive);
	fbP1040Table.p_bSliderActive	:= ADR(tyP1040Table.bSliderActive);
	fbP1040Table;

	//Table Content
	IF tyP1040Table.bTableActive = TRUE OR tyP1040Table.bSliderActive = TRUE OR bRefreshProdRcpTable = TRUE OR bUpdateP1040Table THEN
		FOR i := 1 TO c_uiP1040TableSize DO
			IF tyP1040ProdSet.tyProdSet.tyBtnSort.bValue THEN
				tyP1040ProdSet.tyProdSet.tyTableRecipe.a_tyStringDataCol0[i].sValue	    := UINT_TO_STRING(tyP1040Table.uiTablePos + i - 1);
				tyP1040ProdSet.tyProdSet.tyTableRecipe.a_tyStringDataCol1[i].sValue		:= p_tyProdRcpSortedList[tyP1040Table.uiTablePos + i - 1].sRcpNm;
				tyP1040ProdSet.tyProdSet.tyTableRecipe.a_tyStringDataCol2[i].sValue		:= p_tyProdRcpSortedList[tyP1040Table.uiTablePos + i - 1].sDisplayInfo;
			ELSE

			IF tyP1040ProdSet.tyProdSet.tyStringSearch.sValue = '' THEN
				tyP1040ProdSet.tyProdSet.tyTableRecipe.a_tyStringDataCol0[i].sValue	:= UINT_TO_STRING(tyP1040Table.uiTablePos + i - 1);
				tyP1040ProdSet.tyProdSet.tyTableRecipe.a_tyStringDataCol1[i].sValue	:= p_tyProdRcpCurrList[tyP1040Table.uiTablePos + i - 1].sRcpNm;
				tyP1040ProdSet.tyProdSet.tyTableRecipe.a_tyStringDataCol2[i].sValue	:= p_tyProdRcpCurrList[tyP1040Table.uiTablePos + i - 1].sDisplayInfo;
			ELSE
				tyP1040ProdSet.tyProdSet.tyTableRecipe.a_tyStringDataCol0[i].sValue	:= UINT_TO_STRING(tyP1040Table.uiTablePos + i - 1);
				tyP1040ProdSet.tyProdSet.tyTableRecipe.a_tyStringDataCol1[i].sValue	:= p_tyProdRcpFilterList[tyP1040Table.uiTablePos + i - 1].sRcpNm;
				tyP1040ProdSet.tyProdSet.tyTableRecipe.a_tyStringDataCol2[i].sValue	:= p_tyProdRcpFilterList[tyP1040Table.uiTablePos + i - 1].sDisplayInfo;
				END_IF
			END_IF

		END_FOR

		IF bUpdateP1040Table THEN
			bUpdateP1040Table := FALSE;
		END_IF
	END_IF

	//Selected Row
	IF tyP1040Table.uiSelectedRow <> tyP1040Table.uiSelectedRowOld THEN

		FOR i := 1 TO c_uiP1040TableSize DO

			IF tyP1040Table.uiSelectedRow = i THEN
				tyP1040ProdSet.tyProdSet.tyTableRecipe.a_tyStringDataCol1[i].usiColor	:= 1;
				tyP1040ProdSet.tyProdSet.tyTableRecipe.a_tyStringDataCol2[i].usiColor	:= 1;
			ELSE
				tyP1040ProdSet.tyProdSet.tyTableRecipe.a_tyStringDataCol1[i].usiColor	:= 0;
				tyP1040ProdSet.tyProdSet.tyTableRecipe.a_tyStringDataCol2[i].usiColor	:= 0;
			END_IF

		END_FOR

		tyP1040Table.uiSelectedRowOld	:= tyP1040Table.uiSelectedRow;

	END_IF

END_ACTION
```

#### Act_OptP1040Search.st
```iecst
ACTION Act_OptP1040Search:

	//Search Input Valid
	IF tyP1040ProdSet.tyProdSet.tyStringSearch.bRtCompl = TRUE THEN

		IF tyP1040ProdSet.tyProdSet.tyStringSearch.sValue = '' THEN

			FOR i := 1 TO c_uiP1040TableSize DO
				tyP1040ProdSet.tyProdSet.tyTableRecipe.a_tyStringDataCol0[i].sValue	:= UINT_TO_STRING(tyP1040Table.uiTablePos + i - 1);
				tyP1040ProdSet.tyProdSet.tyTableRecipe.a_tyStringDataCol1[i].sValue	:= p_tyProdRcpCurrList[tyP1040Table.uiTablePos + i - 1].sRcpNm;
				tyP1040ProdSet.tyProdSet.tyTableRecipe.a_tyStringDataCol2[i].sValue	:= p_tyProdRcpCurrList[tyP1040Table.uiTablePos + i - 1].sDisplayInfo;
			END_FOR

			tyP1040ProdSet.tyProdSet.tyStringSearch.bRtCompl	:= FALSE;
			bRefreshProdRcpDetail								:= TRUE;

			IF tyP1040ProdSet.tyProdSet.tyBtnSort.bValue THEN
				bFilterSortP1040	:= TRUE;
			END_IF

		ELSE

			tyP1040ProdSet.tyProdSet.tyTableRecipe.uiMaskRtStat	:= FALSE;
			tyP1040ProdSet.tyProdSet.tyBtnSave.uiMaskRtStat		:= FALSE;
			tyP1040ProdSet.tyProdSet.tyBtnDelete.uiMaskRtStat	:= FALSE;

			sProdRcpSearch	:= tyP1040ProdSet.tyProdSet.tyStringSearch.sValue;

			eProdRcpAct	:= ProdRcpActFilter;

			IF p_eProdRcpStat = ProdRcpActFilter AND p_eProdRcpStatus = Done THEN
				eProdRcpAct	:= ProdRcpActIdle;

				FOR i := 1 TO c_uiP1040TableSize DO
					tyP1040ProdSet.tyProdSet.tyTableRecipe.a_tyStringDataCol0[i].sValue	:= UINT_TO_STRING(tyP1040Table.uiTablePos + i - 1);
					tyP1040ProdSet.tyProdSet.tyTableRecipe.a_tyStringDataCol1[i].sValue	:= p_tyProdRcpFilterList[tyP1040Table.uiTablePos + i - 1].sRcpNm;
					tyP1040ProdSet.tyProdSet.tyTableRecipe.a_tyStringDataCol2[i].sValue	:= p_tyProdRcpFilterList[tyP1040Table.uiTablePos + i - 1].sDisplayInfo;
				END_FOR

				//Unmask Table
				tyP1040ProdSet.tyProdSet.tyTableRecipe.uiMaskRtStat	:= TRUE;
				tyP1040ProdSet.tyProdSet.tyBtnSave.uiMaskRtStat		:= FALSE;
				tyP1040ProdSet.tyProdSet.tyBtnDelete.uiMaskRtStat	:= TRUE;

				//Reset
				tyP1040ProdSet.tyProdSet.tyStringSearch.bRtCompl	:= FALSE;
				bRefreshProdRcpDetail								:= TRUE;

				IF tyP1040ProdSet.tyProdSet.tyBtnSort.bValue THEN
					bFilterSortP1040	:= TRUE;
				END_IF

			ELSIF p_eProdRcpStatus = Error THEN

				FOR i := 1 TO c_uiP1040TableSize DO
					tyP1040ProdSet.tyProdSet.tyTableRecipe.a_tyStringDataCol0[i].sValue	:= UINT_TO_STRING(tyP1040Table.uiTablePos + i - 1);
					tyP1040ProdSet.tyProdSet.tyTableRecipe.a_tyStringDataCol1[i].sValue	:= '';
					tyP1040ProdSet.tyProdSet.tyTableRecipe.a_tyStringDataCol2[i].sValue	:= '';
				END_FOR

				p_tyC0008MsgBox ACCESS ADR (tyP1040ProdSet.tyMsgBoxListErr);

				IF tyP1040ProdSet.tyMsgBoxListErr.tyBtnNo.bRtCompl = TRUE THEN
					tyP1040ProdSet.tyMsgBoxListErr.tyBtnNo.bRtCompl	:= TRUE;
					tyP1040ProdSet.tyMsgBoxListErr.tyBtnNo.bValue	:= TRUE;

					p_tyC0008MsgBox ACCESS ADR (tyP1040ProdSet.tyMsgBoxHide);

					//Unmask Table
					tyP1040ProdSet.tyProdSet.tyTableRecipe.uiMaskRtStat	:= TRUE;
					tyP1040ProdSet.tyProdSet.tyBtnSave.uiMaskRtStat		:= FALSE;
					tyP1040ProdSet.tyProdSet.tyBtnDelete.uiMaskRtStat	:= TRUE;

					//Reset
					tyP1040ProdSet.tyProdSet.tyStringSearch.bRtCompl	:= FALSE;
					bRefreshProdRcpDetail								:= TRUE;
				END_IF

			END_IF

		END_IF

	END_IF

END_ACTION
```

#### Act_OptP1040Keypad.st
```iecst
ACTION Act_OptP1040Keypad:

	IF fUIOutRtStatTPIsOpen(ADR(tyP1040ProdSet.tyProdSet.tyStringRecipeNm.uiRtStat)) THEN
		tyProperty.tyKeypad.tyTxtTitle.sTxt	:= tyP1040ProdSet.tyProdSet.tyStringRecipeNm.sKeypadTitle;

	ELSIF fUIOutRtStatTPIsOpen(ADR(tyP1040ProdSet.tyProdSet.tyNumProdWidth.uiRtStat)) THEN
		IF p_tyNtParamCurr.bLFProdWidth2Prep THEN
			tyProperty.tyKeypad.tyTxtTitle.sTxt	:= 'Product Width US';
		ELSE
			tyProperty.tyKeypad.tyTxtTitle.sTxt	:= 'Product Width DS';
		END_IF

	ELSIF fUIOutRtStatTPIsOpen(ADR(tyP1040ProdSet.tyProdSet.tyNumProdWidth2.uiRtStat)) THEN
		tyProperty.tyKeypad.tyTxtTitle.sTxt	:='Product Width DS';

	ELSIF fUIOutRtStatTPIsOpen(ADR(tyP1040ProdSet.tyProdSet.tyNumProdWidth.uiRtStat)) THEN
		tyProperty.tyKeypad.tyTxtTitle.sTxt	:= tyP1040ProdSet.tyProdSet.tyNumProdWidth.sKeypadTitle;

	ELSIF fUIOutRtStatTPIsOpen(ADR(tyP1040ProdSet.tyProdSet.tyStringSearch.uiRtStat)) THEN
		tyProperty.tyKeypad.tyTxtTitle.sTxt	:= tyP1040ProdSet.tyProdSet.tyStringSearch.sKeypadTitle;

	ELSIF fUIOutRtStatTPIsOpen(ADR(tyP1040ProdSet.tyProdSet.tyStringMatchCode.uiRtStat)) THEN
		tyProperty.tyKeypad.tyTxtTitle.sTxt	:= tyP1040ProdSet.tyProdSet.tyStringMatchCode.sKeypadTitle;

	END_IF

END_ACTION
```

#### Act_OptP1040Sort.st
```iecst
ACTION Act_OptP1040Sort:

	IF tyP1040ProdSet.tyProdSet.tyBtnSort.bValue THEN
		tyP1040ProdSet.tyProdSet.tyBtnSort.usiTxtIdx 	:= 1;

	ELSE
		tyP1040ProdSet.tyProdSet.tyBtnSort.usiTxtIdx 	:= 0;

	END_IF

	IF tyP1040ProdSet.tyProdSet.tyBtnSort.bRtCompl THEN
		bUpdateP1040LoadData := TRUE;
	END_IF

	IF tyP1040ProdSet.tyProdSet.tyBtnSort.bRtCompl OR (bFilterSortP1040 AND p_eProdRcpStat<> ProdRcpActFilter) THEN

		IF tyP1040ProdSet.tyProdSet.tyBtnSort.bValue THEN

			tyP1040ProdSet.tyProdSet.tyTableRecipe.uiMaskRtStat.0	:= FALSE;

			sProdRcpSearch	:= tyP1040ProdSet.tyProdSet.tyStringSearch.sValue;

			eProdRcpAct	:= ProdRcpActSort;

			IF p_eProdRcpStat = ProdRcpActSort AND p_eProdRcpStatus = Done THEN
				eProdRcpAct		:= ProdRcpActIdle;

				FOR i := 1 TO c_uiP1040TableSize DO
					tyP1040ProdSet.tyProdSet.tyTableRecipe.a_tyStringDataCol0[i].sValue	:= UINT_TO_STRING(tyP1040Table.uiTablePos + i - 1);
					tyP1040ProdSet.tyProdSet.tyTableRecipe.a_tyStringDataCol1[i].sValue	:= p_tyProdRcpSortedList[tyP1040Table.uiTablePos + i - 1].sRcpNm;
					tyP1040ProdSet.tyProdSet.tyTableRecipe.a_tyStringDataCol2[i].sValue	:= p_tyProdRcpSortedList[tyP1040Table.uiTablePos + i - 1].sDisplayInfo;
				END_FOR

				bFilterSortP1040	:= FALSE;

				//Unmask
				tyP1040ProdSet.tyProdSet.tyTableRecipe.uiMaskRtStat.0	:= TRUE;

				tyP1040ProdSet.tyProdSet.tyBtnSort.bRtCompl := FALSE;

			ELSIF p_eProdRcpStatus = Error THEN
				FOR i := 1 TO c_uiP1040TableSize DO
					tyP1040ProdSet.tyProdSet.tyTableRecipe.a_tyStringDataCol0[i].sValue		:= UINT_TO_STRING(tyP1040Table.uiTablePos + i - 1);
					tyP1040ProdSet.tyProdSet.tyTableRecipe.a_tyStringDataCol1[i].sValue		:= '';
					tyP1040ProdSet.tyProdSet.tyTableRecipe.a_tyStringDataCol2[i].sValue		:= '';
				END_FOR

				p_tyC0008MsgBox ACCESS ADR (tyP1040ProdSet.tyMsgBoxListErr);

				bFilterSortP1040	:= FALSE;

				IF tyP1040ProdSet.tyMsgBoxListErr.tyBtnNo.bRtCompl = TRUE THEN
					tyP1040ProdSet.tyMsgBoxListErr.tyBtnNo.bRtCompl 		:= TRUE;
					tyP1040ProdSet.tyMsgBoxListErr.tyBtnNo.bValue			:= TRUE;

					p_tyC0008MsgBox ACCESS ADR (tyP1040ProdSet.tyMsgBoxHide);

					//Unmask
					tyP1040ProdSet.tyProdSet.tyTableRecipe.uiMaskRtStat.0	:= TRUE;

					//Reset
					tyP1040ProdSet.tyProdSet.tyBtnSort.bRtCompl := FALSE;
				END_IF
			END_IF

		ELSE

			bUpdateP1040Table	:= TRUE;

			tyP1040ProdSet.tyProdSet.tyBtnSort.bRtCompl := FALSE;

		END_IF

	END_IF

END_ACTION
```

#### Act_OptP1040ToXML.st
```iecst
ACTION Act_OptP1040ToXML:

	IF tyP1040ProdSet.tyProdSet.tyBtnToXML.bRtCompl = TRUE THEN

		IF usiProdRcpToXMLStep = 0 THEN
			//Confirmation Message - To XML Ask
			//Mask
			fUIInRtStatOff(ADR(tyP1040ProdSet.tyProdSet.tyStringSearch.uiMaskRtStat));
			fUIInRtStatOff(ADR(tyP1040ProdSet.tyProdSet.tyTableRecipe.uiMaskRtStat));

			p_tyC0008MsgBox ACCESS ADR(tyP1040ProdSet.tyMsgBoxToXMLAsk);

			IF tyP1040ProdSet.tyMsgBoxToXMLAsk.tyBtnYes.bRtCompl = TRUE THEN
				tyP1040ProdSet.tyMsgBoxToXMLAsk.tyBtnYes.bRtCompl	:= FALSE;
				tyP1040ProdSet.tyMsgBoxToXMLAsk.tyBtnYes.bValue		:= FALSE;

				p_tyC0008MsgBox ACCESS ADR(tyP1040ProdSet.tyMsgBoxHide);

				usiProdRcpToXMLStep	:= 1;

			ELSIF tyP1040ProdSet.tyMsgBoxToXMLAsk.tyBtnNo.bRtCompl = TRUE THEN
				tyP1040ProdSet.tyMsgBoxToXMLAsk.tyBtnNo.bRtCompl	:= FALSE;
				tyP1040ProdSet.tyMsgBoxToXMLAsk.tyBtnNo.bValue		:= FALSE;

				p_tyC0008MsgBox ACCESS ADR(tyP1040ProdSet.tyMsgBoxHide);

				usiProdRcpToXMLStep	:= 99;
			END_IF

		ELSIF usiProdRcpToXMLStep = 1 THEN
			//Save Recipe To XML
			eMpProdRcpAct	:= MpProdRcpActSave;

			IF p_eMpProdRcpStat = MpProdRcpActSave AND p_eMpProdRcpStatus = Done THEN
				eMpProdRcpAct	:= MpProdRcpActIdle;

				tyP1040ProdSet.tyProdSet.tyBtnSort.bValue := FALSE;
				tyP1040ProdSet.tyProdSet.tyStringSearch.sValue := '';
				bRefreshProdRcpTable	:= TRUE;
				bRefreshProdRcpDetail	:= TRUE;

				usiProdRcpToXMLStep		:= 99;

			ELSIF p_eMpProdRcpStatus = Error THEN
				p_tyC0008MsgBox ACCESS ADR(tyP1040ProdSet.tyMsgBoxToXMLErr);

				IF tyP1040ProdSet.tyMsgBoxToXMLErr.tyBtnNo.bRtCompl = TRUE THEN
					tyP1040ProdSet.tyMsgBoxToXMLErr.tyBtnNo.bRtCompl	:= FALSE;
					tyP1040ProdSet.tyMsgBoxToXMLErr.tyBtnNo.bValue		:= FALSE;

					p_tyC0008MsgBox ACCESS ADR(tyP1040ProdSet.tyMsgBoxHide);

					usiProdRcpToXMLStep	:= 99;
				END_IF

			END_IF

		ELSIF usiProdRcpToXMLStep = 99 THEN
			//Complete Reset
			bRefreshProdRcpTable	:= FALSE;

			//Unmask
			fUIInRtStatHide(ADR(tyP1040ProdSet.tyProdSet.tyStringSearch.uiMaskRtStat));
			fUIInRtStatHide(ADR(tyP1040ProdSet.tyProdSet.tyTableRecipe.uiMaskRtStat));

			tyP1040ProdSet.tyProdSet.tyBtnToXML.bRtCompl	:= FALSE;
			tyP1040ProdSet.tyProdSet.tyBtnToXML.bValue		:= FALSE;

			usiProdRcpToXMLStep	:= 0;

		END_IF

	END_IF

END_ACTION
```

#### Act_OptP1040FromXML.st
```iecst
ACTION Act_OptP1040FromXML:

	IF tyP1040ProdSet.tyProdSet.tyBtnFromXML.bRtCompl = TRUE THEN

		IF usiProdRcpFromXMLStep = 0 THEN
			//Confirmation Message - From XML Ask
			//Mask
			fUIInRtStatOff(ADR(tyP1040ProdSet.tyProdSet.tyStringSearch.uiMaskRtStat));
			fUIInRtStatOff(ADR(tyP1040ProdSet.tyProdSet.tyTableRecipe.uiMaskRtStat));

			p_tyC0008MsgBox ACCESS ADR(tyP1040ProdSet.tyMsgBoxFromXMLAsk);

			IF tyP1040ProdSet.tyMsgBoxFromXMLAsk.tyBtnYes.bRtCompl = TRUE THEN
				tyP1040ProdSet.tyMsgBoxFromXMLAsk.tyBtnYes.bRtCompl	:= FALSE;
				tyP1040ProdSet.tyMsgBoxFromXMLAsk.tyBtnYes.bValue	:= FALSE;

				p_tyC0008MsgBox ACCESS ADR(tyP1040ProdSet.tyMsgBoxHide);

				usiProdRcpFromXMLStep	:= 1;

			ELSIF tyP1040ProdSet.tyMsgBoxFromXMLAsk.tyBtnNo.bRtCompl = TRUE THEN
				tyP1040ProdSet.tyMsgBoxFromXMLAsk.tyBtnNo.bRtCompl	:= FALSE;
				tyP1040ProdSet.tyMsgBoxFromXMLAsk.tyBtnNo.bValue	:= FALSE;

				p_tyC0008MsgBox ACCESS ADR(tyP1040ProdSet.tyMsgBoxHide);

				usiProdRcpFromXMLStep	:= 99;
			END_IF

		ELSIF usiProdRcpFromXMLStep = 1 THEN
			//Load Recipe From XML
			eMpProdRcpAct	:= MpProdRcpActLoad;

			IF p_eMpProdRcpStat = MpProdRcpActLoad AND p_eMpProdRcpStatus = Done THEN
				eMpProdRcpAct	:= MpProdRcpActIdle;

				tyP1040ProdSet.tyProdSet.tyBtnSort.bValue := FALSE;
				tyP1040ProdSet.tyProdSet.tyStringSearch.sValue := '';
				bRefreshProdRcpTable	:= TRUE;
				bRefreshProdRcpDetail	:= TRUE;

				usiProdRcpFromXMLStep	:= 2;

			ELSIF p_eMpProdRcpStatus = Error THEN
				p_tyC0008MsgBox ACCESS ADR(tyP1040ProdSet.tyMsgBoxFromXMLErr);

				IF tyP1040ProdSet.tyMsgBoxFromXMLErr.tyBtnNo.bRtCompl = TRUE THEN
					tyP1040ProdSet.tyMsgBoxFromXMLErr.tyBtnNo.bRtCompl	:= FALSE;
					tyP1040ProdSet.tyMsgBoxFromXMLErr.tyBtnNo.bValue	:= FALSE;

					p_tyC0008MsgBox ACCESS ADR(tyP1040ProdSet.tyMsgBoxHide);

					usiProdRcpFromXMLStep	:= 99;
				END_IF

			END_IF

		ELSIF usiProdRcpFromXMLStep = 2 THEN
			//Save Product Recipe List
			eProdRcpAct	:= ProdRcpActSaveList;

			IF p_eProdRcpStat = ProdRcpActSaveList AND p_eProdRcpStatus = Done THEN
				eProdRcpAct	:= ProdRcpActIdle;

				usiProdRcpFromXMLStep	:= 99;

			ELSIF p_eProdRcpStatus = Error THEN
				p_tyC0008MsgBox ACCESS ADR(tyP1040ProdSet.tyMsgBoxSaveListErr);

				IF tyP1040ProdSet.tyMsgBoxSaveListErr.tyBtnNo.bRtCompl = TRUE THEN
					tyP1040ProdSet.tyMsgBoxSaveListErr.tyBtnNo.bRtCompl	:= FALSE;
					tyP1040ProdSet.tyMsgBoxSaveListErr.tyBtnNo.bValue	:= FALSE;

					p_tyC0008MsgBox ACCESS ADR(tyP1040ProdSet.tyMsgBoxHide);

					usiProdRcpFromXMLStep	:= 99;
				END_IF

			END_IF

		ELSIF usiProdRcpFromXMLStep = 99 THEN
			//Complete Reset
			bRefreshProdRcpTable	:= FALSE;

			//Unmask
			fUIInRtStatHide(ADR(tyP1040ProdSet.tyProdSet.tyStringSearch.uiMaskRtStat));
			fUIInRtStatHide(ADR(tyP1040ProdSet.tyProdSet.tyTableRecipe.uiMaskRtStat));

			tyP1040ProdSet.tyProdSet.tyBtnFromXML.bRtCompl	:= FALSE;
			tyP1040ProdSet.tyProdSet.tyBtnFromXML.bValue	:= FALSE;

			usiProdRcpFromXMLStep	:= 0;

		END_IF

	END_IF

END_ACTION
```

#### Act_OptP1040RcpPopUp.st
```iecst
ACTION Act_OptP1040RcpPopUp:

	tyP1040ProdSet.tyProdSet.tyHotspotShowLRcp.uiRtStat.0	:= NOT(tyP1040ProdSet.tyProdSet.tyStringRecipeNm.sValue <> '');

	IF tyP1040ProdSet.tyProdSet.tyHotspotShowLRcp.bRtCompl = TRUE THEN
		tyP1040ProdSet.tyProdSet.tyHotspotShowLRcp.bRtCompl  := FALSE;

		fUIInRtStatOff(ADR(tyP1040ProdSet.tyRcpPopUp.tyLyr.uiRtStat));

		tyP1040ProdSet.tyRcpPopUp.tyStringInfo.sValue  :=  tyP1040ProdSet.tyProdSet.tyStringRecipeNm.sValue; // Show 254 Characters

	ELSIF tyP1040ProdSet.tyRcpPopUp.tyHotspotClose.bRtCompl = TRUE THEN
		tyP1040ProdSet.tyRcpPopUp.tyHotspotClose.bRtCompl := FALSE;

		fUIInRtStatHide(ADR(tyP1040ProdSet.tyRcpPopUp.tyLyr.uiRtStat)); // Hide Pop Up Again

	END_IF

END_ACTION
```

#### Act_EntP1050Disp.st
```iecst
ACTION Act_EntP1050Disp:

	//Access Address
	p_tyC0005Main ACCESS ADR(tyCommon.tyMain);

	p_tyC0006Set ACCESS ADR(tyCommon.tySet);

	p_tyC0007Notif ACCESS ADR(tyCommon.tyNotif);

	p_tyC0008MsgBox ACCESS ADR(tyP1050LFSet.tyMsgBoxHide);

	p_tyC0009Info ACCESS ADR(tyCommon.tyInfo);

	p_tyC0011Loading ACCESS ADR(tyCommon.tyLoading);

	p_tyP1050LFSetLdrEdit ACCESS ADR(tyP1050LFSet.tyLdrEdit);

	p_tyP1050LFSetLdr ACCESS ADR(tyP1050LFSet.tyLdr);

END_ACTION
```

#### Act_OptP1050Edit.st
```iecst
ACTION Act_OptP1050Edit:

	IF tyP1050LFSet.tyLdr.tyBtnEdit.bRtCompl = TRUE THEN

		FOR i := 1 TO UDINT_TO_UINT(c_diLFClntNum) DO
			IF tyMcParamWr.a_sLFIPAddr[i] = '' THEN
				uiLFStartEditNo	:= i;
				EXIT;
			END_IF
		END_FOR

		tyP1050LFSet.tyLdr.tyBtnEdit.bRtCompl	:= FALSE;
		tyP1050LFSet.tyLdr.tyBtnEdit.bValue		:= TRUE;

		fUIInRtStatOff(ADR(tyP1050LFSet.tyLdrEdit.tyLyr.uiRtStat));
		fUIInRtStatHide(ADR(tyP1050LFSet.tyLdr.tyLyr.uiRtStat));

		tyP1050LFSet.tyLdrEdit.tyNumMcNum.diValue		:= STRING_TO_DINT(tyP1050LFSet.tyLdr.tyTable1List.a_tyStringDataCol0[tyP1050Table.uiSelectedRow].sValue);
		tyP1050LFSet.tyLdrEdit.tyStringIPAddr.sValue	:= tyP1050LFSet.tyLdr.tyTable1List.a_tyStringDataCol2[tyP1050Table.uiSelectedRow].sValue;

	ELSIF tyP1050LFSet.tyLdr.tyBtnEdit.bValue = TRUE THEN

		IF tyP1050LFSet.tyLdrEdit.tyBtnOk.bRtCompl = TRUE THEN

			IF fIPValid(tyP1050LFSet.tyLdrEdit.tyStringIPAddr.sValue , ADR(a_iIPPart1)) = TRUE AND bCheckDone = FALSE THEN
				FOR i := 1 TO UDINT_TO_UINT(c_diLFClntNum) DO
					IF i <>  tyP1050Table.uiTablePos + tyP1050Table.uiSelectedRow - 1 THEN
						fIPValid(p_tyMcParamCurr.a_sLFIPAddr[i] , ADR(a_iIPPart2));

						IF (a_iIPPart1[1] = a_iIPPart2[1] AND a_iIPPart1[2] = a_iIPPart2[2] AND a_iIPPart1[3] = a_iIPPart2[3] AND a_iIPPart1[4] = a_iIPPart2[4])
							AND (tyP1050LFSet.tyLdrEdit.tyStringIPAddr.sValue <> '') THEN

							bIPDuplicate	:= TRUE;
							EXIT;

						END_IF
					END_IF
				END_FOR
				bCheckDone := TRUE;
			END_IF

			IF fIPValid(tyP1050LFSet.tyLdrEdit.tyStringIPAddr.sValue , ADR(a_iIPPart1)) = FALSE THEN
				p_tyC0008MsgBox ACCESS ADR(tyP1050LFSet.tyMsgBoxIPAddrInvalid);

				IF tyP1050LFSet.tyMsgBoxIPAddrInvalid.tyBtnNo.bRtCompl = TRUE THEN
					tyP1050LFSet.tyMsgBoxIPAddrInvalid.tyBtnNo.bRtCompl	:= FALSE;
					tyP1050LFSet.tyMsgBoxIPAddrInvalid.tyBtnNo.bValue	:= FALSE;

					p_tyC0008MsgBox ACCESS ADR(tyP1050LFSet.tyMsgBoxHide);

					tyP1050LFSet.tyLdrEdit.tyBtnOk.bRtCompl	:= FALSE;
					tyP1050LFSet.tyLdrEdit.tyBtnOk.bValue	:= FALSE;
					bCheckDone := FALSE;
				END_IF

			ELSIF bIPDuplicate = TRUE THEN
				p_tyC0008MsgBox ACCESS ADR(tyP1050LFSet.tyMsgBoxIPAddrDuplicate);

				IF tyP1050LFSet.tyMsgBoxIPAddrDuplicate.tyBtnNo.bRtCompl = TRUE THEN
					tyP1050LFSet.tyMsgBoxIPAddrDuplicate.tyBtnNo.bRtCompl	:= FALSE;
					tyP1050LFSet.tyMsgBoxIPAddrDuplicate.tyBtnNo.bValue		:= FALSE;

					p_tyC0008MsgBox ACCESS ADR(tyP1050LFSet.tyMsgBoxHide);

					bIPDuplicate							:= FALSE;
					tyP1050LFSet.tyLdrEdit.tyBtnOk.bRtCompl	:= FALSE;
					tyP1050LFSet.tyLdrEdit.tyBtnOk.bValue	:= FALSE;
					bCheckDone := FALSE;
				END_IF
			ELSE
				tyMcParamWr.a_sLFIPAddr[tyP1050Table.uiTablePos + tyP1050Table.uiSelectedRow - 1]	:= tyP1050LFSet.tyLdrEdit.tyStringIPAddr.sValue;

				eMcParamAct	:= McParamActWrite;

				IF p_eMcParamStat = McParamActWrite AND p_eMcParamStatus = Done THEN
					eMcParamAct	:= McParamActIdle;

					tyP1050LFSet.tyLdr.tyTable1List.a_tyStringDataCol2[tyP1050Table.uiSelectedRow].sValue		:= tyP1050LFSet.tyLdrEdit.tyStringIPAddr.sValue;

					IF tyP1050LFSet.tyLdrEdit.tyStringIPAddr.sValue = '0000' THEN
						tyP1050LFSet.tyLdr.tyTable1List.a_tyTxtDataCol3[tyP1050Table.uiSelectedRow].usiValueIdx	:= 3;
					ELSE
						tyP1050LFSet.tyLdr.tyTable1List.a_tyTxtDataCol3[tyP1050Table.uiSelectedRow].usiValueIdx	:= 1;
					END_IF

					//LF Control
					FOR i := 1 TO c_uiP1050TableSize DO
						tyP0700LFCtrl.tyLdr.tyTable1List.a_tyStringDataCol0[i].sValue	:= UINT_TO_STRING(tyP0700Table.uiTablePos + i - 1);
						tyP0700LFCtrl.tyLdr.tyTable1List.a_tyStringDataCol2[i].sValue	:= p_tyMcParamCurr.a_sLFIPAddr[tyP0700Table.uiTablePos + i - 1];
					END_FOR

					tyP1050LFSet.tyLdrEdit.tyBtnOk.bRtCompl	:= FALSE;
					tyP1050LFSet.tyLdrEdit.tyBtnOk.bValue	:= FALSE;
					tyP1050LFSet.tyLdr.tyBtnEdit.bValue		:= FALSE;
					bCheckDone								:= FALSE;

					fUIInRtStatHide(ADR(tyP1050LFSet.tyLdrEdit.tyLyr.uiRtStat));
					fUIInRtStatOff(ADR(tyP1050LFSet.tyLdr.tyLyr.uiRtStat));

				ELSIF p_eMcParamStatus = Error THEN
					p_tyC0008MsgBox ACCESS ADR(tyP1050LFSet.tyMsgBoxSaveErr);

					IF tyP1050LFSet.tyMsgBoxSaveErr.tyBtnNo.bRtCompl = TRUE THEN
						tyP1050LFSet.tyMsgBoxSaveErr.tyBtnNo.bRtCompl	:= FALSE;
						tyP1050LFSet.tyMsgBoxSaveErr.tyBtnNo.bValue		:= FALSE;

						p_tyC0008MsgBox ACCESS ADR(tyP1050LFSet.tyMsgBoxHide);

						//Recover
						tyMcParamWr	:= p_tyMcParamCurr;

						tyP1050LFSet.tyLdrEdit.tyBtnOk.bRtCompl	:= FALSE;
						tyP1050LFSet.tyLdrEdit.tyBtnOk.bValue	:= FALSE;
						tyP1050LFSet.tyLdr.tyBtnEdit.bValue		:= FALSE;
						bCheckDone								:=FALSE;

						fUIInRtStatHide(ADR(tyP1050LFSet.tyLdrEdit.tyLyr.uiRtStat));
						fUIInRtStatOff(ADR(tyP1050LFSet.tyLdr.tyLyr.uiRtStat));
					END_IF
				END_IF
			END_IF
		ELSIF tyP1050LFSet.tyLdrEdit.tyBtnCancel.bRtCompl = TRUE THEN
			tyP1050LFSet.tyLdrEdit.tyBtnCancel.bRtCompl	:= FALSE;
			tyP1050LFSet.tyLdrEdit.tyBtnCancel.bValue	:= FALSE;
			tyP1050LFSet.tyLdr.tyBtnEdit.bValue			:= FALSE;

			fUIInRtStatHide(ADR(tyP1050LFSet.tyLdrEdit.tyLyr.uiRtStat));
			fUIInRtStatOff(ADR(tyP1050LFSet.tyLdr.tyLyr.uiRtStat));
		END_IF
	END_IF

	IF bLFSettingAutoFill THEN

		iIPExtract:= LEN(p_sHWInfoIPAddr)-10;
		sLFSettingCurrentIP := RIGHT(p_sHWInfoIPAddr,iIPExtract);
		iLFSettingCurrentIP	:= STRING_TO_INT(sLFSettingCurrentIP);

		FOR i:= 1 TO 20 DO
			sLFSettingAutoFill	:='192.168.0.';
			sLFSettingTemp		:=UINT_TO_STRING(iLFSettingCurrentIP+(i*2)-2);
			sLFSettingAutoFill	:=CONCAT(sLFSettingAutoFill,sLFSettingTemp);
			tyMcParamWr.a_sLFIPAddr[i]:= sLFSettingAutoFill;
			tyMcParamWr.a_bLFOnline[i]:= FALSE;
		END_FOR

		eMcParamAct	:= McParamActWrite;

		IF p_eMcParamStat = McParamActWrite AND p_eMcParamStatus = Done THEN
			eMcParamAct	:= McParamActIdle;
			bUpdateP1050Table	:= TRUE;
			bLFSettingAutoFill	:= FALSE;
		ELSIF p_eMcParamStatus = Error THEN
			//Recover
			tyMcParamWr	:= p_tyMcParamCurr;
			bUpdateP1050Table	:= TRUE;
			bLFSettingAutoFill	:= FALSE;
		END_IF

	END_IF

	IF bLFSettingAutoClear THEN
		FOR i:= 1 TO 20 DO
			tyMcParamWr.a_sLFIPAddr[i]:= '';
			tyMcParamWr.a_bLFOnline[i]:= FALSE;
		END_FOR

		eMcParamAct	:= McParamActWrite;

		IF p_eMcParamStat = McParamActWrite AND p_eMcParamStatus = Done THEN
			eMcParamAct	:= McParamActIdle;
			bUpdateP1050Table	:= TRUE;
			bLFSettingAutoClear	:= FALSE;
		ELSIF p_eMcParamStatus = Error THEN
			//Recover
			tyMcParamWr	:= p_tyMcParamCurr;
			bUpdateP1050Table	:= TRUE;
			bLFSettingAutoClear	:= FALSE;
		END_IF

	END_IF

END_ACTION
```

#### Act_OptP1050Online.st
```iecst
ACTION Act_OptP1050Online:

	IF tyP1050LFSet.tyLdr.tyBtnOnline.bRtCompl = TRUE THEN
		tyMcParamWr.a_bLFOnline[tyP1050Table.uiTablePos + tyP1050Table.uiSelectedRow - 1]	:= TRUE;

		eMcParamAct	:= McParamActWrite;

		IF p_eMcParamStat = McParamActWrite AND p_eMcParamStatus = Done THEN
			eMcParamAct	:= McParamActIdle;

			tyP1050LFSet.tyLdr.tyTable1List.a_tyTxtDataCol3[tyP1050Table.uiSelectedRow].usiValueIdx	:= 2;

			//Reset
			tyP1050LFSet.tyLdr.tyBtnOnline.bRtCompl		:= FALSE;
			tyP1050LFSet.tyLdr.tyBtnOnline.bValue		:= FALSE;

		ELSIF p_eMcParamStatus = Error THEN
			p_tyC0008MsgBox ACCESS ADR(tyP1050LFSet.tyMsgBoxSaveErr);

			IF tyP1050LFSet.tyMsgBoxSaveErr.tyBtnNo.bRtCompl = TRUE THEN
				tyP1050LFSet.tyMsgBoxSaveErr.tyBtnNo.bRtCompl	:= FALSE;
				tyP1050LFSet.tyMsgBoxSaveErr.tyBtnNo.bValue		:= FALSE;

				p_tyC0008MsgBox ACCESS ADR(tyP1050LFSet.tyMsgBoxHide);

				//Recover
				tyMcParamWr	:= p_tyMcParamCurr;

				//Reset
				tyP1050LFSet.tyLdr.tyBtnOnline.bRtCompl	:= FALSE;
				tyP1050LFSet.tyLdr.tyBtnOnline.bValue	:= FALSE;
			END_IF
		END_IF
	END_IF

END_ACTION
```

#### Act_OptP1050Offline.st
```iecst
ACTION Act_OptP1050Offline:

	IF tyP1050LFSet.tyLdr.tyBtnOffline.bRtCompl = TRUE THEN
		tyMcParamWr.a_bLFOnline[tyP1050Table.uiTablePos + tyP1050Table.uiSelectedRow - 1]	:= FALSE;

		eMcParamAct	:= McParamActWrite;

		IF p_eMcParamStat = McParamActWrite AND p_eMcParamStatus = Done THEN
			eMcParamAct	:= McParamActIdle;

			tyP1050LFSet.tyLdr.tyTable1List.a_tyTxtDataCol3[tyP1050Table.uiSelectedRow].usiValueIdx	:= 1;

			//Reset
			tyP1050LFSet.tyLdr.tyBtnOffline.bRtCompl	:= FALSE;
			tyP1050LFSet.tyLdr.tyBtnOffline.bValue		:= FALSE;

		ELSIF p_eMcParamStatus = Error THEN
			p_tyC0008MsgBox ACCESS ADR(tyP1050LFSet.tyMsgBoxSaveErr);

			IF tyP1050LFSet.tyMsgBoxSaveErr.tyBtnNo.bRtCompl = TRUE THEN
				tyP1050LFSet.tyMsgBoxSaveErr.tyBtnNo.bRtCompl	:= FALSE;
				tyP1050LFSet.tyMsgBoxSaveErr.tyBtnNo.bValue		:= FALSE;

				p_tyC0008MsgBox ACCESS ADR(tyP1050LFSet.tyMsgBoxHide);

				//Recover
				tyMcParamWr	:= p_tyMcParamCurr;

				//Reset
				tyP1050LFSet.tyLdr.tyBtnOffline.bRtCompl	:= FALSE;
				tyP1050LFSet.tyLdr.tyBtnOffline.bValue		:= FALSE;
			END_IF
		END_IF
	END_IF

END_ACTION
```

#### Act_OptP1050Delete.st
```iecst
ACTION Act_OptP1050Delete:

	IF tyP1050LFSet.tyLdr.tyBtnDelete.bRtCompl = TRUE THEN

		IF usiDelMcDetailsStep = 0 THEN
			p_tyC0008MsgBox ACCESS ADR(tyP1050LFSet.tyMsgBoxDelAsk);

			IF tyP1050LFSet.tyMsgBoxDelAsk.tyBtnYes.bRtCompl = TRUE THEN
				tyP1050LFSet.tyMsgBoxDelAsk.tyBtnYes.bRtCompl	:= FALSE;
				tyP1050LFSet.tyMsgBoxDelAsk.tyBtnYes.bValue		:= FALSE;

				p_tyC0008MsgBox ACCESS ADR(tyP1050LFSet.tyMsgBoxHide);

				usiDelMcDetailsStep	:= 1;

			ELSIF tyP1050LFSet.tyMsgBoxDelAsk.tyBtnNo.bRtCompl = TRUE THEN
				tyP1050LFSet.tyMsgBoxDelAsk.tyBtnNo.bRtCompl	:= FALSE;
				tyP1050LFSet.tyMsgBoxDelAsk.tyBtnNo.bValue		:= FALSE;

				p_tyC0008MsgBox ACCESS ADR(tyP1050LFSet.tyMsgBoxHide);

				tyP1050LFSet.tyLdr.tyBtnDelete.bRtCompl			:= FALSE;
				tyP1050LFSet.tyLdr.tyBtnDelete.bValue			:= FALSE;
			END_IF

		ELSIF usiDelMcDetailsStep = 1 THEN
//			tyMcParamWr.a_sLFIPAddr[tyP1050Table.uiTablePos + tyP1050Table.uiSelectedRow - 1]	:= '';
//			tyMcParamWr.a_bLFOnline[tyP1050Table.uiTablePos + tyP1050Table.uiSelectedRow - 1]	:= FALSE;

			IF bLFDeleteOn=FALSE THEN

				memcpy(ADR(tyMcParamWr.a_sLFIPAddr[tyP1050Table.uiTablePos + tyP1050Table.uiSelectedRow - 1]),ADR(tyMcParamWr.a_sLFIPAddr[tyP1050Table.uiTablePos + tyP1050Table.uiSelectedRow]),(SIZEOF(tyMcParamWr.a_sLFIPAddr[1]) * (50-(tyP1050Table.uiTablePos + tyP1050Table.uiSelectedRow-1))));
				memset(ADR(tyMcParamWr.a_sLFIPAddr[50]),0,SIZEOF(tyMcParamWr.a_sLFIPAddr[1]));

				memcpy(ADR(tyMcParamWr.a_bLFOnline[tyP1050Table.uiTablePos + tyP1050Table.uiSelectedRow - 1]),ADR(tyMcParamWr.a_bLFOnline[tyP1050Table.uiTablePos + tyP1050Table.uiSelectedRow]),(SIZEOF(tyMcParamWr.a_bLFOnline[1]) * (50-(tyP1050Table.uiTablePos + tyP1050Table.uiSelectedRow-1))));
				memset(ADR(tyMcParamWr.a_bLFOnline[50]),0,SIZEOF(tyMcParamWr.a_bLFOnline[1]));

				bLFDeleteOn:= TRUE;

			END_IF

			eMcParamAct	:= McParamActWrite;

			IF p_eMcParamStat = McParamActWrite AND p_eMcParamStatus = Done THEN
				eMcParamAct	:= McParamActIdle;

				tyP1050LFSet.tyLdr.tyTable1List.a_tyStringDataCol2[tyP1050Table.uiSelectedRow].sValue	:= '';
				tyP1050LFSet.tyLdr.tyTable1List.a_tyTxtDataCol3[tyP1050Table.uiSelectedRow].usiValueIdx	:= 0;

				//P0700 LF Control
				FOR i := 1 TO c_uiP1050TableSize DO
					tyP0700LFCtrl.tyLdr.tyTable1List.a_tyStringDataCol0[i].sValue	:= UINT_TO_STRING(tyP0700Table.uiTablePos + i - 1);
					tyP0700LFCtrl.tyLdr.tyTable1List.a_tyStringDataCol2[i].sValue	:= p_tyMcParamCurr.a_sLFIPAddr[tyP0700Table.uiTablePos + i - 1];
				END_FOR

				usiDelMcDetailsStep	:= 0;

				tyP1050LFSet.tyLdr.tyBtnDelete.bRtCompl	:= FALSE;
				tyP1050LFSet.tyLdr.tyBtnDelete.bValue	:= FALSE;

				bLFDeleteOn			:=FALSE;
				bUpdateP1050Table	:=TRUE;

			ELSIF p_eMcParamStatus = Error THEN
				p_tyC0008MsgBox ACCESS ADR(tyP1050LFSet.tyMsgBoxSaveErr);

				bLFDeleteOn			:=FALSE;

				IF tyP1050LFSet.tyMsgBoxSaveErr.tyBtnNo.bRtCompl = TRUE THEN
					tyP1050LFSet.tyMsgBoxSaveErr.tyBtnNo.bRtCompl	:= FALSE;
					tyP1050LFSet.tyMsgBoxSaveErr.tyBtnNo.bValue		:= FALSE;

					p_tyC0008MsgBox ACCESS ADR(tyP1050LFSet.tyMsgBoxHide);

					//Recover
					tyMcParamWr	:= p_tyMcParamCurr;

					usiDelMcDetailsStep	:= 0;

					tyP1050LFSet.tyLdr.tyBtnDelete.bRtCompl	:= FALSE;
					tyP1050LFSet.tyLdr.tyBtnDelete.bValue	:= FALSE;
				END_IF

			END_IF

		END_IF

	END_IF

END_ACTION
```

#### Act_OptP1050Mask.st
```iecst
ACTION Act_OptP1050Mask:

	IF tyP1050LFSet.tyLdr.tyBtnOnline.bRtCompl THEN
		tyP1050LFSet.tyLdr.tyBtnEdit.uiMaskRtStat					:= FALSE;
		tyP1050LFSet.tyLdr.tyBtnOffline.uiMaskRtStat				:= FALSE;
		tyP1050LFSet.tyLdr.tyBtnDelete.uiMaskRtStat					:= FALSE;
		tyP1050LFSet.tyLdr.tyBtnShftUp.uiMaskRtStat					:= FALSE;
		tyP1050LFSet.tyLdr.tyBtnShftDwn.uiMaskRtStat				:= FALSE;
		tyP1050LFSet.tyLdr.tyTable1List.uiMaskRtStat				:= FALSE;

	ELSIF tyP1050LFSet.tyLdr.tyBtnOffline.bRtCompl THEN
		tyP1050LFSet.tyLdr.tyBtnEdit.uiMaskRtStat					:= FALSE;
		tyP1050LFSet.tyLdr.tyBtnOnline.uiMaskRtStat					:= FALSE;
		tyP1050LFSet.tyLdr.tyBtnDelete.uiMaskRtStat					:= FALSE;
		tyP1050LFSet.tyLdr.tyBtnShftUp.uiMaskRtStat					:= FALSE;
		tyP1050LFSet.tyLdr.tyBtnShftDwn.uiMaskRtStat				:= FALSE;
		tyP1050LFSet.tyLdr.tyTable1List.uiMaskRtStat				:= FALSE;

	ELSIF tyP1050LFSet.tyLdr.tyBtnDelete.bRtCompl THEN
		tyP1050LFSet.tyLdr.tyBtnEdit.uiMaskRtStat					:= FALSE;
		tyP1050LFSet.tyLdr.tyBtnOnline.uiMaskRtStat					:= FALSE;
		tyP1050LFSet.tyLdr.tyBtnOffline.uiMaskRtStat				:= FALSE;
		tyP1050LFSet.tyLdr.tyBtnShftUp.uiMaskRtStat					:= FALSE;
		tyP1050LFSet.tyLdr.tyBtnShftDwn.uiMaskRtStat				:= FALSE;
		tyP1050LFSet.tyLdr.tyTable1List.uiMaskRtStat				:= FALSE;

	ELSIF tyP1050LFSet.tyLdr.tyBtnShftUp.bRtCompl THEN
		tyP1050LFSet.tyLdr.tyBtnEdit.uiMaskRtStat					:= FALSE;
		tyP1050LFSet.tyLdr.tyBtnOnline.uiMaskRtStat					:= FALSE;
		tyP1050LFSet.tyLdr.tyBtnOffline.uiMaskRtStat				:= FALSE;
		tyP1050LFSet.tyLdr.tyBtnDelete.uiMaskRtStat					:= FALSE;
		tyP1050LFSet.tyLdr.tyBtnShftDwn.uiMaskRtStat				:= FALSE;
		tyP1050LFSet.tyLdr.tyTable1List.uiMaskRtStat				:= FALSE;

	ELSIF tyP1050LFSet.tyLdr.tyBtnShftDwn.bRtCompl THEN
		tyP1050LFSet.tyLdr.tyBtnEdit.uiMaskRtStat					:= FALSE;
		tyP1050LFSet.tyLdr.tyBtnOnline.uiMaskRtStat					:= FALSE;
		tyP1050LFSet.tyLdr.tyBtnOffline.uiMaskRtStat				:= FALSE;
		tyP1050LFSet.tyLdr.tyBtnDelete.uiMaskRtStat					:= FALSE;
		tyP1050LFSet.tyLdr.tyBtnShftUp.uiMaskRtStat					:= FALSE;
		tyP1050LFSet.tyLdr.tyTable1List.uiMaskRtStat				:= FALSE;

	ELSE
		tyP1050LFSet.tyLdr.tyBtnEdit.uiMaskRtStat					:= TRUE;
		tyP1050LFSet.tyLdr.tyTable1List.uiMaskRtStat				:= TRUE;

		IF tyP1050LFSet.tyLdr.tyTable1List.a_tyStringDataCol2[tyP1050Table.uiSelectedRow].sValue = '' THEN
			tyP1050LFSet.tyLdr.tyBtnOnline.uiMaskRtStat				:= FALSE;
			tyP1050LFSet.tyLdr.tyBtnOffline.uiMaskRtStat			:= FALSE;
			tyP1050LFSet.tyLdr.tyBtnDelete.uiMaskRtStat				:= FALSE;
			tyP1050LFSet.tyLdr.tyBtnShftUp.uiMaskRtStat				:= FALSE;
			tyP1050LFSet.tyLdr.tyBtnShftDwn.uiMaskRtStat			:= FALSE;

		ELSE
			tyP1050LFSet.tyLdr.tyBtnDelete.uiMaskRtStat				:= TRUE;

			IF tyP1050LFSet.tyLdr.tyTable1List.a_tyStringDataCol2[tyP1050Table.uiSelectedRow].sValue = '0000' THEN
				tyP1050LFSet.tyLdr.tyBtnOnline.uiMaskRtStat			:= FALSE;
				tyP1050LFSet.tyLdr.tyBtnOffline.uiMaskRtStat		:= FALSE;

			ELSE
				IF tyP1050LFSet.tyLdr.tyTable1List.a_tyTxtDataCol3[tyP1050Table.uiSelectedRow].usiValueIdx = 2 THEN
					tyP1050LFSet.tyLdr.tyBtnOnline.uiMaskRtStat		:= FALSE;
					tyP1050LFSet.tyLdr.tyBtnOffline.uiMaskRtStat	:= TRUE;
				ELSE
					tyP1050LFSet.tyLdr.tyBtnOnline.uiMaskRtStat		:= TRUE;
					tyP1050LFSet.tyLdr.tyBtnOffline.uiMaskRtStat	:= FALSE;
				END_IF

			END_IF

			//Shift Up
			IF tyP1050Table.uiSelectedRow = 1 AND tyP1050LFSet.tyLdr.tyTable1List.a_tyStringDataCol0[1].sValue = '1' THEN
				tyP1050LFSet.tyLdr.tyBtnShftUp.uiMaskRtStat			:= FALSE;
			ELSE
				tyP1050LFSet.tyLdr.tyBtnShftUp.uiMaskRtStat			:= TRUE;
			END_IF

			//Shift Down
			IF tyP1050Table.uiSelectedRow = c_uiP1050TableSize AND STRING_TO_UINT(tyP1050LFSet.tyLdr.tyTable1List.a_tyStringDataCol0[c_uiP1050TableSize].sValue) = c_diLFClntNum THEN
				tyP1050LFSet.tyLdr.tyBtnShftDwn.uiMaskRtStat		:= FALSE;
			ELSE
				IF tyP1050LFSet.tyLdr.tyTable1List.a_tyStringDataCol2[tyP1050Table.uiSelectedRow+1].sValue = '' THEN
					tyP1050LFSet.tyLdr.tyBtnShftDwn.uiMaskRtStat		:= FALSE;
				ELSE
					tyP1050LFSet.tyLdr.tyBtnShftDwn.uiMaskRtStat		:= TRUE;
				END_IF
			END_IF

		END_IF

	END_IF

END_ACTION
```

#### Act_OptP1050Table.st
```iecst
ACTION Act_OptP1050Table:

	//Call Table FB
	fbP1050Table.sVisuNm			:= tyP1050Table.sVisuNm;
	fbP1050Table.udiWorkAreaStartX	:= 96;
	fbP1050Table.udiWorkAreaEndX	:= 554;
	fbP1050Table.udiWorkAreaStartY	:= 75;
	fbP1050Table.udiWorkAreaEndY	:= 455;
	fbP1050Table.udiMinXDist		:= 20;
	fbP1050Table.udiMinYDist		:= 20;
	fbP1050Table.uiSlideScale		:= c_uiP1050TableSize;
	fbP1050Table.iTotalData			:= UDINT_TO_INT(c_diLFClntNum);
	fbP1050Table.iTotalRow			:= c_uiP1050TableSize;
	fbP1050Table(uiSliderStatus := tyP1050LFSet.tyLdr.tyTable1List.tyUISlider.uiRtStat , a_tyUIHotspot := tyP1050LFSet.tyLdr.tyTable1List.a_tyHotspot , uiTablePos := tyP1050Table.uiTablePos , iSliderPos := tyP1050LFSet.tyLdr.tyTable1List.tyUISlider.iValue);

	tyP1050Table.uiSelectedRow		:= fbP1050Table.uiSelectedRow;
	tyP1050Table.bTableActive		:= fbP1050Table.bTableActive;
	tyP1050Table.bSliderActive		:= fbP1050Table.bSliderActive;

	//Table Content
	IF tyP1050Table.bTableActive = TRUE OR tyP1050Table.bSliderActive = TRUE OR usiTableShftStep = 3 OR bUpdateP1050Table THEN
		FOR i := 1 TO c_uiP1050TableSize DO
			tyP1050LFSet.tyLdr.tyTable1List.a_tyStringDataCol0[i].sValue			:= UINT_TO_STRING(tyP1050Table.uiTablePos + i - 1);
			tyP1050LFSet.tyLdr.tyTable1List.a_tyStringDataCol2[i].sValue			:= p_tyMcParamCurr.a_sLFIPAddr[tyP1050Table.uiTablePos + i - 1];

			IF tyP1050LFSet.tyLdr.tyTable1List.a_tyStringDataCol2[i].sValue = '' THEN
				tyP1050LFSet.tyLdr.tyTable1List.a_tyTxtDataCol3[i].usiValueIdx	:= 0;
			ELSIF tyP1050LFSet.tyLdr.tyTable1List.a_tyStringDataCol2[i].sValue = '0000' THEN
				tyP1050LFSet.tyLdr.tyTable1List.a_tyTxtDataCol3[i].usiValueIdx	:= 3;
			ELSE
				tyP1050LFSet.tyLdr.tyTable1List.a_tyTxtDataCol3[i].usiValueIdx	:= (BOOL_TO_USINT(p_tyMcParamCurr.a_bLFOnline[tyP1050Table.uiTablePos + i - 1])) + 1;
			END_IF

		END_FOR

		IF bUpdateP1050Table THEN
			bUpdateP1050Table := FALSE;
		END_IF

	END_IF

	//Selected Row
	IF tyP1050Table.uiSelectedRow <> tyP1050Table.uiSelectedRowOld THEN
		FOR i := 1 TO c_uiP1050TableSize DO
			IF tyP1050Table.uiSelectedRow = i THEN
				tyP1050LFSet.tyLdr.tyTable1List.a_tyStringDataCol2[i].usiColor	:= 1;
				tyP1050LFSet.tyLdr.tyTable1List.a_tyTxtDataCol3[i].usiColor		:= 1;

			ELSE
				tyP1050LFSet.tyLdr.tyTable1List.a_tyStringDataCol2[i].usiColor	:= 0;
				tyP1050LFSet.tyLdr.tyTable1List.a_tyTxtDataCol3[i].usiColor		:= 0;

			END_IF

		END_FOR

		tyP1050Table.uiSelectedRowOld	:= tyP1050Table.uiSelectedRow;

	END_IF

END_ACTION
```

#### Act_OptP1050ShftUp.st
```iecst
ACTION Act_OptP1050ShftUp:

	IF tyP1050LFSet.tyLdr.tyBtnShftUp.bRtCompl = TRUE THEN
		IF usiTableShftStep = 0 THEN
			IF tyP1050Table.uiSelectedRow = 1 AND tyP1050LFSet.tyLdr.tyTable1List.a_tyStringDataCol0[1].sValue = '1' THEN
				tyP1050LFSet.tyLdr.tyBtnShftUp.bValue	:= FALSE;
				tyP1050LFSet.tyLdr.tyBtnShftUp.bRtCompl	:= FALSE;
			ELSE
				usiTableShftStep	:= 1;
			END_IF

		ELSIF usiTableShftStep = 1 THEN
			IF p_tyMcParamCurr.a_sLFIPAddr[tyP1050Table.uiTablePos + tyP1050Table.uiSelectedRow - 2] <> '' THEN
				sLFIPAddrTemp	:= p_tyMcParamCurr.a_sLFIPAddr[tyP1050Table.uiTablePos + tyP1050Table.uiSelectedRow - 2];

				tyMcParamWr.a_sLFIPAddr[tyP1050Table.uiTablePos + tyP1050Table.uiSelectedRow - 2]	:= p_tyMcParamCurr.a_sLFIPAddr[tyP1050Table.uiTablePos + tyP1050Table.uiSelectedRow - 1];
				tyMcParamWr.a_sLFIPAddr[tyP1050Table.uiTablePos + tyP1050Table.uiSelectedRow - 1]	:= sLFIPAddrTemp;

				bOnlineTemp		:= p_tyMcParamCurr.a_bLFOnline[tyP1050Table.uiTablePos + tyP1050Table.uiSelectedRow - 2];

				tyMcParamWr.a_bLFOnline[tyP1050Table.uiTablePos + tyP1050Table.uiSelectedRow - 2]	:= p_tyMcParamCurr.a_bLFOnline[tyP1050Table.uiTablePos + tyP1050Table.uiSelectedRow - 1];
				tyMcParamWr.a_bLFOnline[tyP1050Table.uiTablePos + tyP1050Table.uiSelectedRow - 1]	:= bOnlineTemp;
			ELSE
				tyMcParamWr.a_sLFIPAddr[tyP1050Table.uiTablePos + tyP1050Table.uiSelectedRow - 2]	:= p_tyMcParamCurr.a_sLFIPAddr[tyP1050Table.uiTablePos + tyP1050Table.uiSelectedRow - 1];
				memset(ADR(tyMcParamWr.a_sLFIPAddr[tyP1050Table.uiTablePos + tyP1050Table.uiSelectedRow - 1]), 0, SIZEOF(tyMcParamWr.a_sLFIPAddr[tyP1050Table.uiTablePos + tyP1050Table.uiSelectedRow - 1]));

				tyMcParamWr.a_bLFOnline[tyP1050Table.uiTablePos + tyP1050Table.uiSelectedRow - 2]	:= p_tyMcParamCurr.a_bLFOnline[tyP1050Table.uiTablePos + tyP1050Table.uiSelectedRow - 1];
				tyMcParamWr.a_bLFOnline[tyP1050Table.uiTablePos + tyP1050Table.uiSelectedRow - 1]	:= FALSE;
			END_IF

			usiTableShftStep	:= 2;

		ELSIF usiTableShftStep = 2 THEN
			eMcParamAct	:= McParamActWrite;

			IF p_eMcParamStat = McParamActWrite AND p_eMcParamStatus = Done THEN
				eMcParamAct	:= McParamActIdle;

				//Table
				IF tyP1050Table.uiSelectedRow <> 1 THEN
					fbP1050Table.bSelectedRowMnl	:= TRUE;
					fbP1050Table.uiSelectedRowMnl	:= tyP1050Table.uiSelectedRow - 1;
				ELSE
					fbP1050Table.bTablePosMinus		:= TRUE;
				END_IF

				usiTableShftStep	:= 3;

			ELSIF p_eMcParamStatus = Error THEN
				p_tyC0008MsgBox ACCESS ADR(tyP1050LFSet.tyMsgBoxSaveErr);

				IF tyP1050LFSet.tyMsgBoxSaveErr.tyBtnNo.bRtCompl = TRUE THEN
					tyP1050LFSet.tyMsgBoxSaveErr.tyBtnNo.bRtCompl	:= FALSE;
					tyP1050LFSet.tyMsgBoxSaveErr.tyBtnNo.bValue		:= FALSE;

					p_tyC0008MsgBox ACCESS ADR(tyP1050LFSet.tyMsgBoxHide);

					//Recover
					tyMcParamWr	:= p_tyMcParamCurr;

					usiTableShftStep	:= 0;

					tyP1050LFSet.tyLdr.tyBtnShftUp.bRtCompl	:= FALSE;
					tyP1050LFSet.tyLdr.tyBtnShftUp.bValue	:= FALSE;
				END_IF
			END_IF

		ELSIF usiTableShftStep = 3 THEN
			//UIP0700 LF Control
			FOR i := 1 TO c_uiP0700TableSize DO
				tyP0700LFCtrl.tyLdr.tyTable1List.a_tyStringDataCol0[i].sValue	:= UINT_TO_STRING(tyP0700Table.uiTablePos + i - 1);
				tyP0700LFCtrl.tyLdr.tyTable1List.a_tyStringDataCol2[i].sValue	:= p_tyMcParamCurr.a_sLFIPAddr[tyP0700Table.uiTablePos + i - 1];
			END_FOR

			//Rst Table Control
			fbP1050Table.bSelectedRowMnl	:= FALSE;
			fbP1050Table.bTablePosMinus		:= FALSE;

			usiTableShftStep	:= 0;

			tyP1050LFSet.tyLdr.tyBtnShftUp.bRtCompl	:= FALSE;
			tyP1050LFSet.tyLdr.tyBtnShftUp.bValue	:= FALSE;
		END_IF
	END_IF

END_ACTION
```

#### Act_OptP1050ShftDwn.st
```iecst
ACTION Act_OptP1050ShftDwn:

	IF tyP1050LFSet.tyLdr.tyBtnShftDwn.bRtCompl = TRUE THEN
		IF usiTableShftStep = 0 THEN
			IF tyP1050Table.uiSelectedRow = c_uiP1050TableSize AND STRING_TO_UINT(tyP1050LFSet.tyLdr.tyTable1List.a_tyStringDataCol0[c_uiP1050TableSize].sValue) = c_diLFClntNum THEN
				tyP1050LFSet.tyLdr.tyBtnShftDwn.bValue	:= FALSE;
				tyP1050LFSet.tyLdr.tyBtnShftDwn.bRtCompl:= FALSE;
			ELSE
				usiTableShftStep	:= 1;
			END_IF

		ELSIF usiTableShftStep = 1 THEN
			IF p_tyMcParamCurr.a_sLFIPAddr[tyP1050Table.uiTablePos + tyP1050Table.uiSelectedRow] <> '' THEN
				sLFIPAddrTemp	:= p_tyMcParamCurr.a_sLFIPAddr[tyP1050Table.uiTablePos + tyP1050Table.uiSelectedRow];

				tyMcParamWr.a_sLFIPAddr[tyP1050Table.uiTablePos + tyP1050Table.uiSelectedRow]		:= p_tyMcParamCurr.a_sLFIPAddr[tyP1050Table.uiTablePos + tyP1050Table.uiSelectedRow - 1];
				tyMcParamWr.a_sLFIPAddr[tyP1050Table.uiTablePos + tyP1050Table.uiSelectedRow - 1]	:= sLFIPAddrTemp;

				bOnlineTemp		:= p_tyMcParamCurr.a_bLFOnline[tyP1050Table.uiTablePos + tyP1050Table.uiSelectedRow];

				tyMcParamWr.a_bLFOnline[tyP1050Table.uiTablePos + tyP1050Table.uiSelectedRow]		:= p_tyMcParamCurr.a_bLFOnline[tyP1050Table.uiTablePos + tyP1050Table.uiSelectedRow - 1];
				tyMcParamWr.a_bLFOnline[tyP1050Table.uiTablePos + tyP1050Table.uiSelectedRow - 1]	:= bOnlineTemp;

			ELSE
				tyMcParamWr.a_sLFIPAddr[tyP1050Table.uiTablePos + tyP1050Table.uiSelectedRow]		:= p_tyMcParamCurr.a_sLFIPAddr[tyP1050Table.uiTablePos + tyP1050Table.uiSelectedRow - 1];
				memset(ADR(tyMcParamWr.a_sLFIPAddr[tyP1050Table.uiTablePos + tyP1050Table.uiSelectedRow - 1]), 0, SIZEOF(tyMcParamWr.a_sLFIPAddr[tyP1050Table.uiTablePos + tyP1050Table.uiSelectedRow - 1]));

				tyMcParamWr.a_bLFOnline[tyP1050Table.uiTablePos + tyP1050Table.uiSelectedRow]		:= p_tyMcParamCurr.a_bLFOnline[tyP1050Table.uiTablePos + tyP1050Table.uiSelectedRow - 1];
				tyMcParamWr.a_bLFOnline[tyP1050Table.uiTablePos + tyP1050Table.uiSelectedRow - 1]	:= FALSE;
			END_IF

			usiTableShftStep	:= 2;

		ELSIF usiTableShftStep = 2 THEN
			eMcParamAct	:= McParamActWrite;

			IF p_eMcParamStat = McParamActWrite AND p_eMcParamStatus = Done THEN
				eMcParamAct	:= McParamActIdle;

				//Table
				IF tyP1050Table.uiSelectedRow <> c_uiP1050TableSize THEN
					fbP1050Table.bSelectedRowMnl	:= TRUE;
					fbP1050Table.uiSelectedRowMnl	:= tyP1050Table.uiSelectedRow + 1;
				ELSE
					fbP1050Table.bTablePosPlus		:= TRUE;
				END_IF

				usiTableShftStep	:= 3;

			ELSIF p_eMcParamStatus = Error THEN
				p_tyC0008MsgBox ACCESS ADR(tyP1050LFSet.tyMsgBoxSaveErr);

				IF tyP1050LFSet.tyMsgBoxSaveErr.tyBtnNo.bRtCompl = TRUE THEN
					tyP1050LFSet.tyMsgBoxSaveErr.tyBtnNo.bRtCompl	:= FALSE;
					tyP1050LFSet.tyMsgBoxSaveErr.tyBtnNo.bValue		:= FALSE;

					p_tyC0008MsgBox ACCESS ADR(tyP1050LFSet.tyMsgBoxHide);

					//Recover
					tyMcParamWr	:= p_tyMcParamCurr;

					usiTableShftStep	:= 0;

					tyP1050LFSet.tyLdr.tyBtnShftDwn.bRtCompl:= FALSE;
					tyP1050LFSet.tyLdr.tyBtnShftDwn.bValue	:= FALSE;
				END_IF
			END_IF

		ELSIF usiTableShftStep = 3 THEN
			//UIP0700 LF Control
			FOR i := 1 TO c_uiP0700TableSize DO
				tyP0700LFCtrl.tyLdr.tyTable1List.a_tyStringDataCol0[i].sValue	:= UINT_TO_STRING(tyP0700Table.uiTablePos + i - 1);
				tyP0700LFCtrl.tyLdr.tyTable1List.a_tyStringDataCol2[i].sValue	:= p_tyMcParamCurr.a_sLFIPAddr[tyP0700Table.uiTablePos + i - 1];
			END_FOR

			//Rst Table Control
			fbP1050Table.bSelectedRowMnl	:= FALSE;
			fbP1050Table.bTablePosPlus		:= FALSE;

			usiTableShftStep	:= 0;

			tyP1050LFSet.tyLdr.tyBtnShftDwn.bRtCompl:= FALSE;
			tyP1050LFSet.tyLdr.tyBtnShftDwn.bValue	:= FALSE;
		END_IF
	END_IF

END_ACTION
```

#### Act_OptP1050Keypad.st
```iecst
ACTION Act_OptP1050Keypad:

	IF fUIOutRtStatTPIsOpen(ADR(tyP1050LFSet.tyLdrEdit.tyStringIPAddr.uiRtStat)) THEN
		tyProperty.tyKeypad.tyTxtTitle.sTxt	:= tyP1050LFSet.tyLdrEdit.tyStringIPAddr.sKeypadTitle;

	ELSIF fUIOutRtStatTPIsOpen(ADR(tyP1050LFSet.tyLdr.tyNumAfterOven.uiRtStat)) THEN
		tyProperty.tyKeypad.tyTxtTitle.sTxt	:= tyP1050LFSet.tyLdr.tyNumAfterOven.sKeypadTitle;

	ELSIF fUIOutRtStatTPIsOpen(ADR(tyP1050LFSet.tyLdr.tyNumBeforeOven.uiRtStat)) THEN
		tyProperty.tyKeypad.tyTxtTitle.sTxt	:= tyP1050LFSet.tyLdr.tyNumBeforeOven.sKeypadTitle;

	ELSIF fUIOutRtStatTPIsOpen(ADR(tyP1050LFSet.tyLdr.tyNumAfterOven2.uiRtStat)) THEN
		tyProperty.tyKeypad.tyTxtTitle.sTxt	:= tyP1050LFSet.tyLdr.tyNumAfterOven2.sKeypadTitle;

	ELSIF fUIOutRtStatTPIsOpen(ADR(tyP1050LFSet.tyLdr.tyNumBeforeOven2.uiRtStat)) THEN
		tyProperty.tyKeypad.tyTxtTitle.sTxt	:= tyP1050LFSet.tyLdr.tyNumBeforeOven2.sKeypadTitle;

	ELSE
		tyProperty.tyKeypad.tyTxtTitle.sTxt	:= '';

	END_IF

END_ACTION
```

#### Act_OptP1050Oven.st
```iecst
ACTION Act_OptP1050Oven:

	IF tyP1050LFSet.tyLdr.tyNumBeforeOven.bRtCompl = TRUE	OR tyP1050LFSet.tyLdr.tyNumAfterOven.bRtCompl = TRUE
		OR tyP1050LFSet.tyLdr.tyNumBeforeOven2.bRtCompl = TRUE	OR tyP1050LFSet.tyLdr.tyNumAfterOven2.bRtCompl = TRUE THEN

		tyMcParamWr.diLFMcIdxBeforeOven		:= tyP1050LFSet.tyLdr.tyNumBeforeOven.diValue;
		tyMcParamWr.diLFMcIdxAfterOven		:= tyP1050LFSet.tyLdr.tyNumAfterOven.diValue;
		tyMcParamWr.diLFMcIdxBeforeOven2	:= tyP1050LFSet.tyLdr.tyNumBeforeOven2.diValue;
		tyMcParamWr.diLFMcIdxAfterOven2		:= tyP1050LFSet.tyLdr.tyNumAfterOven2.diValue;

		eMcParamAct	:= McParamActWrite;

		IF p_eMcParamStat = McParamActWrite AND p_eMcParamStatus = Done THEN
			eMcParamAct	:= McParamActIdle;

			//BackUp Param
			tyP1050LFSet.tyLdrBkUp	:= tyP1050LFSet.tyLdr;

			tyP1050LFSet.tyLdr.tyNumBeforeOven.bRtCompl		:= FALSE;
			tyP1050LFSet.tyLdr.tyNumAfterOven.bRtCompl		:= FALSE;
			tyP1050LFSet.tyLdr.tyNumBeforeOven2.bRtCompl	:= FALSE;
			tyP1050LFSet.tyLdr.tyNumAfterOven2.bRtCompl		:= FALSE;

		ELSIF p_eMcParamStatus = Error THEN
			p_tyC0008MsgBox ACCESS ADR(tyP1050LFSet.tyMsgBoxSaveErr);

			IF tyP1050LFSet.tyMsgBoxSaveErr.tyBtnNo.bRtCompl = TRUE THEN
				tyP1050LFSet.tyMsgBoxSaveErr.tyBtnNo.bRtCompl	:= FALSE;
				tyP1050LFSet.tyMsgBoxSaveErr.tyBtnNo.bValue		:= FALSE;

				tyP1050LFSet.tyLdr.tyNumBeforeOven.bRtCompl		:= FALSE;
				tyP1050LFSet.tyLdr.tyNumAfterOven.bRtCompl		:= FALSE;
				tyP1050LFSet.tyLdr.tyNumBeforeOven2.bRtCompl	:= FALSE;
				tyP1050LFSet.tyLdr.tyNumAfterOven2.bRtCompl		:= FALSE;

				p_tyC0008MsgBox ACCESS ADR(tyP1050LFSet.tyMsgBoxHide);

				//Restore Param
				tyP1050LFSet.tyLdr	:= tyP1050LFSet.tyLdrBkUp;
				tyMcParamWr			:= p_tyMcParamCurr;
			END_IF

		END_IF

	END_IF

END_ACTION
```

#### Act_EntP1080Disp.st
```iecst
ACTION Act_EntP1080Disp:

	//Access Address
	p_tyC0005Main ACCESS ADR(tyCommon.tyMain);

	p_tyC0007Notif ACCESS ADR(tyCommon.tyNotif);

	p_tyC0008MsgBox ACCESS ADR(tyP1080UsrMgmt.tyMsgBoxHide);

	p_tyC0009Info ACCESS ADR(tyCommon.tyInfo);

	p_tyC0011Loading ACCESS ADR(tyCommon.tyLoading);

	p_tyP1080UsrMgmt ACCESS ADR(tyP1080UsrMgmt.tyUsrMgmt);

	p_tyP1080UsrMgmtAct ACCESS ADR(tyP1080UsrMgmt.tyCreate);

	fUIInRtStatHide(ADR(tyP1080UsrMgmt.tyCreate.tyLyr.uiRtStat));
	fUIInRtStatOff(ADR(tyP1080UsrMgmt.tyUsrMgmt.tyLyr.uiRtStat));

	//Display
	IF tyP1080UsrMgmt.tyUsrMgmt.tyDrpDnLvl.usiValueIdx > tyP1080UsrMgmt.tyUsrMgmt.tyDrpDnLvl.usiValueMaxIdx THEN
		tyP1080UsrMgmt.tyUsrMgmt.tyDrpDnLvl.usiValueIdx			:= 0;
		tyP1080UsrMgmt.tyUsrMgmt.tyDrpDnLvl.bRtCompl			:= TRUE;
	END_IF

END_ACTION
```

#### Act_ExitP1080.st
```iecst
ACTION Act_ExitP1080:

	tyP1080UsrMgmt.tyUsrMgmt.tyBtnNewUsr.bValue			:= FALSE;
	tyP1080UsrMgmt.tyUsrMgmt.tyBtnNewUsr.bRtCompl		:= FALSE;

	tyP1080UsrMgmt.tyUsrMgmt.tyBtnEditDetail.bValue		:= FALSE;
	tyP1080UsrMgmt.tyUsrMgmt.tyBtnEditDetail.bRtCompl	:= FALSE;

	tyP1080UsrMgmt.tyUsrMgmt.tyBtnDeleteUsr.bValue		:= FALSE;
	tyP1080UsrMgmt.tyUsrMgmt.tyBtnDeleteUsr.bRtCompl	:= FALSE;

	usiChgPage	:= 1;

END_ACTION
```

#### Act_OptP1080EditAccess.st
```iecst
ACTION Act_OptP1080EditAccess:

	IF tyP1080UsrMgmt.tyUsrMgmt.tyBtnEditAccess.bRtCompl = TRUE THEN
		tyP1080UsrMgmt.tyUsrMgmt.tyBtnEditAccess.bRtCompl				:= FALSE;
		tyP1080UsrMgmt.tyUsrMgmt.tyBtnEditAccess.bValue					:= FALSE;

		tyP1081UsrMgmtUsrAccessRgt.tyUsrAccessRgtSel.tyDrpDnLevel.bRtCompl := TRUE;

		eChgPage		:= UIP1081UsrMgmtUsrAccessRgt;

	END_IF

END_ACTION
```

#### Act_OptP1080AddUsr.st
```iecst
ACTION Act_OptP1080AddUsr:

	// Add New User Display Control
	IF tyP1080UsrMgmt.tyUsrMgmt.tyBtnNewUsr.bRtCompl = TRUE THEN
		p_tyP1080UsrMgmtAct ACCESS ADR(tyP1080UsrMgmt.tyCreate);

		fUIInRtStatOff(ADR(tyP1080UsrMgmt.tyCreate.tyLyr.uiRtStat));
		fUIInRtStatHide(ADR(tyP1080UsrMgmt.tyUsrMgmt.tyLyr.uiRtStat));

		tyP1080UsrMgmt.tyCreate.tyStringUsrNm.sValue			:= '';
		tyP1080UsrMgmt.tyCreate.tyStringPw.sValue				:= '';
		tyP1080UsrMgmt.tyCreate.tyDrpDnLvl.usiValueIdx			:= 0;

		tyP1080UsrMgmt.tyUsrMgmt.tyBtnNewUsr.bRtCompl			:= FALSE;
		tyP1080UsrMgmt.tyUsrMgmt.tyBtnNewUsr.bValue				:= TRUE;
	END_IF

	// Add New User
	IF tyP1080UsrMgmt.tyUsrMgmt.tyBtnNewUsr.bValue = TRUE THEN
		IF tyP1080UsrMgmt.tyCreate.tyBtnOk.bRtCompl = TRUE THEN
			IF usiSaveUsrMgmtStep = 0 THEN
				tyUsrMgmtInfoIn.sUsrNm			:= tyP1080UsrMgmt.tyCreate.tyStringUsrNm.sValue;
				tyUsrMgmtInfoIn.sPw				:= tyP1080UsrMgmt.tyCreate.tyStringPw.sValue;
				tyUsrMgmtInfoIn.eUsrLvl			:= tyP1080UsrMgmt.tyCreate.tyDrpDnLvl.usiValueIdx + 1;

				eUsrMgmtAct		:= UsrMgmtActAdd;

				IF p_eUsrMgmtStat = UsrMgmtActAdd AND p_eUsrMgmtStatus = Done THEN
					eUsrMgmtAct	:= UsrMgmtActIdle;

					IF p_bUsrMgmtNmEmpty = TRUE THEN
						usiSaveUsrMgmtStep		:= 1;
					ELSIF p_bUsrMgmtListFull = TRUE THEN
						usiSaveUsrMgmtStep		:= 2;
					ELSIF p_bUsrMgmtNmExist = TRUE THEN
						usiSaveUsrMgmtStep		:= 3;
					ELSE
						bRefreshUsrMgmtTable	:= TRUE;
						usiSaveUsrMgmtStep		:= 99;
					END_IF
				ELSIF p_eUsrMgmtStatus = Error THEN
					p_tyC0008MsgBox ACCESS ADR(tyP1080UsrMgmt.tyMsgBoxAddErr);

					IF tyP1080UsrMgmt.tyMsgBoxAddErr.tyBtnNo.bRtCompl = TRUE THEN
						tyP1080UsrMgmt.tyMsgBoxAddErr.tyBtnNo.bRtCompl 			:= FALSE;
						tyP1080UsrMgmt.tyMsgBoxAddErr.tyBtnNo.bValue 			:= FALSE;

						p_tyC0008MsgBox ACCESS ADR(tyP1080UsrMgmt.tyMsgBoxHide);

						usiSaveUsrMgmtStep		:= 99;
					END_IF
				END_IF

			// Recipe No Name
			ELSIF usiSaveUsrMgmtStep = 1 THEN
				p_tyC0008MsgBox ACCESS ADR(tyP1080UsrMgmt.tyMsgBoxAddParamErr);

				IF tyP1080UsrMgmt.tyMsgBoxAddParamErr.tyBtnNo.bRtCompl = TRUE THEN
					tyP1080UsrMgmt.tyMsgBoxAddParamErr.tyBtnNo.bRtCompl 		:= FALSE;
					tyP1080UsrMgmt.tyMsgBoxAddParamErr.tyBtnNo.bValue 			:= FALSE;

					p_tyC0008MsgBox ACCESS ADR(tyP1040ProdSet.tyMsgBoxHide);

					tyP1080UsrMgmt.tyCreate.tyStringUsrNm.sValue				:= '';
					tyP1080UsrMgmt.tyCreate.tyStringPw.sValue					:= '';
					tyP1080UsrMgmt.tyCreate.tyDrpDnLvl.usiValueIdx				:= 0;

					tyP1080UsrMgmt.tyCreate.tyBtnOk.bRtCompl 					:= FALSE;
					tyP1080UsrMgmt.tyCreate.tyBtnOk.bValue 						:= FALSE;

					usiSaveUsrMgmtStep			:= 0;
				END_IF

			// User List Full
			ELSIF usiSaveUsrMgmtStep = 2 THEN
				p_tyC0008MsgBox ACCESS ADR(tyP1080UsrMgmt.tyMsgBoxListFull);

				IF tyP1080UsrMgmt.tyMsgBoxListFull.tyBtnNo.bRtCompl = TRUE THEN
					tyP1080UsrMgmt.tyMsgBoxListFull.tyBtnNo.bRtCompl 			:= FALSE;
					tyP1080UsrMgmt.tyMsgBoxListFull.tyBtnNo.bValue 				:= FALSE;

					p_tyC0008MsgBox ACCESS ADR(tyP1080UsrMgmt.tyMsgBoxHide);

					usiSaveUsrMgmtStep			:= 99;
				END_IF

			// User Name Exist
			ELSIF usiSaveUsrMgmtStep = 3 THEN
				p_tyC0008MsgBox ACCESS ADR(tyP1080UsrMgmt.tyMsgBoxAddNmExist);

				IF tyP1080UsrMgmt.tyMsgBoxAddNmExist.tyBtnNo.bRtCompl = TRUE THEN
					tyP1080UsrMgmt.tyMsgBoxAddNmExist.tyBtnNo.bRtCompl 			:= FALSE;
					tyP1080UsrMgmt.tyMsgBoxAddNmExist.tyBtnNo.bValue 			:= FALSE;

					p_tyC0008MsgBox ACCESS ADR(tyP1040ProdSet.tyMsgBoxHide);

					tyP1080UsrMgmt.tyCreate.tyStringUsrNm.sValue				:= '';
					tyP1080UsrMgmt.tyCreate.tyStringPw.sValue					:= '';
					tyP1080UsrMgmt.tyCreate.tyDrpDnLvl.usiValueIdx				:= 0;

					tyP1080UsrMgmt.tyCreate.tyBtnOk.bRtCompl 					:= FALSE;
					tyP1080UsrMgmt.tyCreate.tyBtnOk.bValue 						:= FALSE;

					usiSaveUsrMgmtStep			:= 0;
				END_IF

			ELSIF usiSaveUsrMgmtStep = 99 THEN
				tyP1080UsrMgmt.tyUsrMgmt.tyBtnNewUsr.bValue						:= FALSE;

				tyP1080UsrMgmt.tyCreate.tyBtnOk.bRtCompl						:= FALSE;
				tyP1080UsrMgmt.tyCreate.tyBtnOk.bValue							:= FALSE;

				tyP1080UsrMgmt.tyCreate.tyStringUsrNm.sValue					:= '';
				tyP1080UsrMgmt.tyCreate.tyStringPw.sValue						:= '';
				tyP1080UsrMgmt.tyCreate.tyDrpDnLvl.usiValueIdx					:= 0;

				usiSaveUsrMgmtStep			:= 0;

				fUIInRtStatOff(ADR(tyP1080UsrMgmt.tyUsrMgmt.tyLyr.uiRtStat));
				fUIInRtStatHide(ADR(tyP1080UsrMgmt.tyCreate.tyLyr.uiRtStat));

			END_IF

		ELSIF tyP1080UsrMgmt.tyCreate.tyBtnCancel.bRtCompl = TRUE THEN
			fUIInRtStatOff(ADR(tyP1080UsrMgmt.tyUsrMgmt.tyLyr.uiRtStat));
			fUIInRtStatHide(ADR(tyP1080UsrMgmt.tyCreate.tyLyr.uiRtStat));

			tyP1080UsrMgmt.tyUsrMgmt.tyBtnNewUsr.bValue							:= FALSE;

			tyP1080UsrMgmt.tyCreate.tyBtnCancel.bRtCompl						:= FALSE;
			tyP1080UsrMgmt.tyCreate.tyBtnCancel.bValue							:= FALSE;
		END_IF

	END_IF

END_ACTION
```

#### Act_OptP1080DelUsr.st
```iecst
ACTION Act_OptP1080DelUsr:

	IF tyP1080UsrMgmt.tyUsrMgmt.tyBtnDeleteUsr.bRtCompl = TRUE THEN
		IF usiDelUsrMgmtStep = 0 THEN
			//Mask
			tyP1080UsrMgmt.tyUsrMgmt.tyBtnNewUsr.uiMaskRtStat					:= FALSE;
			tyP1080UsrMgmt.tyUsrMgmt.tyBtnEditAccess.uiMaskRtStat				:= FALSE;
			tyP1080UsrMgmt.tyUsrMgmt.tyBtnEditDetail.uiMaskRtStat				:= FALSE;
			tyP1080UsrMgmt.tyUsrMgmt.tyTableList.uiMaskRtStat					:= FALSE;

			p_tyC0008MsgBox ACCESS ADR(tyP1080UsrMgmt.tyMsgBoxDelAsk);

			IF tyP1080UsrMgmt.tyMsgBoxDelAsk.tyBtnYes.bRtCompl = TRUE THEN
				tyP1080UsrMgmt.tyMsgBoxDelAsk.tyBtnYes.bRtCompl					:= FALSE;
				tyP1080UsrMgmt.tyMsgBoxDelAsk.tyBtnYes.bValue					:= FALSE;

				p_tyC0008MsgBox ACCESS ADR(tyP1080UsrMgmt.tyMsgBoxHide);

				usiDelUsrMgmtStep			:= 1;

			ELSIF tyP1080UsrMgmt.tyMsgBoxDelAsk.tyBtnNo.bRtCompl = TRUE THEN
				tyP1080UsrMgmt.tyMsgBoxDelAsk.tyBtnNo.bRtCompl					:= FALSE;
				tyP1080UsrMgmt.tyMsgBoxDelAsk.tyBtnNo.bValue					:= FALSE;

				p_tyC0008MsgBox ACCESS ADR(tyP1080UsrMgmt.tyMsgBoxHide);

				usiDelUsrMgmtStep			:= 99;
			END_IF

		ELSIF usiDelUsrMgmtStep = 1 THEN
			tyUsrMgmtInfoIn.sUsrNm			:= tyP1080UsrMgmt.tyUsrMgmt.tyTableList.a_tyStringDataCol1[tyP1080Table.uiSelectedRow].sValue;
			tyUsrMgmtInfoIn.eUsrLvl			:= USINT_TO_UDINT((tyP1080UsrMgmt.tyUsrMgmt.tyTableList.a_tyTxtDataCol3[tyP1080Table.uiSelectedRow].usiValueIdx)- 1);

			eUsrMgmtAct 					:= UsrMgmtActDel;

			IF p_eUsrMgmtStat = UsrMgmtActDel AND p_eUsrMgmtStatus = Done THEN
				eUsrMgmtAct				:= UsrMgmtActIdle;

				IF p_bUsrMgmtUnableDelete = TRUE THEN
					usiDelUsrMgmtStep		:= 2;
				ELSIF p_bUsrMgmtNmEmpty = TRUE THEN
					usiDelUsrMgmtStep		:= 3;
				ELSIF p_bUsrMgmtNmNotExist = TRUE THEN
					usiDelUsrMgmtStep		:= 4;
				ELSE
					bRefreshUsrMgmtTable	:= TRUE;
					usiDelUsrMgmtStep		:= 99;
				END_IF
			END_IF

		ELSIF usiDelUsrMgmtStep = 2 THEN
			p_tyC0008MsgBox ACCESS ADR(tyP1080UsrMgmt.tyMsgBoxDelLastAdminErr);

			IF tyP1080UsrMgmt.tyMsgBoxDelLastAdminErr.tyBtnNo.bRtCompl = TRUE THEN
				tyP1080UsrMgmt.tyMsgBoxDelLastAdminErr.tyBtnNo.bRtCompl 		:= FALSE;
				tyP1080UsrMgmt.tyMsgBoxDelLastAdminErr.tyBtnNo.bValue 			:= FALSE;

				p_tyC0008MsgBox ACCESS ADR(tyP1080UsrMgmt.tyMsgBoxHide);

				usiDelUsrMgmtStep			:= 99;
			END_IF

		// User Managment Param Invalid
		ELSIF usiDelUsrMgmtStep	= 3 THEN
			p_tyC0008MsgBox ACCESS ADR(tyP1080UsrMgmt.tyMsgBoxDelParamErr);

			IF tyP1080UsrMgmt.tyMsgBoxDelParamErr.tyBtnNo.bRtCompl = TRUE THEN
				tyP1080UsrMgmt.tyMsgBoxDelParamErr.tyBtnNo.bRtCompl 			:= FALSE;
				tyP1080UsrMgmt.tyMsgBoxDelParamErr.tyBtnNo.bValue 				:= FALSE;

				p_tyC0008MsgBox ACCESS ADR(tyP1080UsrMgmt.tyMsgBoxHide);

				usiDelUsrMgmtStep			:= 99;
			END_IF

		// Name Not Exist
		ELSIF usiDelUsrMgmtStep = 4 THEN
			p_tyC0008MsgBox ACCESS ADR(tyP1080UsrMgmt.tyMsgBoxDelNmNotExist);

			IF tyP1080UsrMgmt.tyMsgBoxDelNmNotExist.tyBtnNo.bRtCompl = TRUE THEN
				tyP1080UsrMgmt.tyMsgBoxDelNmNotExist.tyBtnNo.bRtCompl 			:= FALSE;
				tyP1080UsrMgmt.tyMsgBoxDelNmNotExist.tyBtnNo.bValue 			:= FALSE;

				p_tyC0008MsgBox ACCESS ADR(tyP1080UsrMgmt.tyMsgBoxHide);

				usiDelUsrMgmtStep			:= 99;
			END_IF

		ELSIF usiDelUsrMgmtStep = 99 THEN
			//Unmask
			tyP1080UsrMgmt.tyUsrMgmt.tyBtnNewUsr.uiMaskRtStat					:= TRUE;
			tyP1080UsrMgmt.tyUsrMgmt.tyBtnEditAccess.uiMaskRtStat				:= TRUE;
			tyP1080UsrMgmt.tyUsrMgmt.tyBtnEditDetail.uiMaskRtStat				:= TRUE;
			tyP1080UsrMgmt.tyUsrMgmt.tyTableList.uiMaskRtStat					:= TRUE;

			//Reset
			tyP1080UsrMgmt.tyUsrMgmt.tyBtnDeleteUsr.bRtCompl					:= FALSE;
			tyP1080UsrMgmt.tyUsrMgmt.tyBtnDeleteUsr.bValue 						:= FALSE;

			usiDelUsrMgmtStep				:= 0;
		END_IF

	END_IF

END_ACTION
```

#### Act_OptP1080EditUsr.st
```iecst
ACTION Act_OptP1080EditUsr:

	// Edit User Display Control
	IF tyP1080UsrMgmt.tyUsrMgmt.tyBtnEditDetail.bRtCompl = TRUE THEN
		p_tyP1080UsrMgmtAct ACCESS ADR(tyP1080UsrMgmt.tyEdit);

		fUIInRtStatOff(ADR(tyP1080UsrMgmt.tyEdit.tyLyr.uiRtStat));
		fUIInRtStatHide(ADR(tyP1080UsrMgmt.tyUsrMgmt.tyLyr.uiRtStat));

		udiP1080SelectedRow		:= STRING_TO_UDINT(tyP1080UsrMgmt.tyUsrMgmt.tyTableList.a_tyStringDataCol0[tyP1080Table.uiSelectedRow].sValue);
		usiP1080SelectedLvl		:= tyP1080UsrMgmt.tyUsrMgmt.tyTableList.a_tyTxtDataCol3[tyP1080Table.uiSelectedRow].usiValueIdx;

		CASE tyP1080UsrMgmt.tyUsrMgmt.tyDrpDnLvl.usiValueIdx OF
			0:
				tyP1080UsrMgmt.tyEdit.tyStringUsrNm.sValue			:= p_tyUsrMgmtAllList[udiP1080SelectedRow].sUsrNm;
				tyP1080UsrMgmt.tyEdit.tyDrpDnLvl.usiValueIdx		:= UDINT_TO_USINT((p_tyUsrMgmtAllList[udiP1080SelectedRow].eUsrLvl) - 1);

			1:
				tyP1080UsrMgmt.tyEdit.tyStringUsrNm.sValue			:= p_tyUsrMgmtLv2List[udiP1080SelectedRow].sUsrNm;
				tyP1080UsrMgmt.tyEdit.tyDrpDnLvl.usiValueIdx		:= UDINT_TO_USINT((p_tyUsrMgmtLv2List[udiP1080SelectedRow].eUsrLvl) - 1);

			2:
				tyP1080UsrMgmt.tyEdit.tyStringUsrNm.sValue			:= p_tyUsrMgmtLv3List[udiP1080SelectedRow].sUsrNm;
				tyP1080UsrMgmt.tyEdit.tyDrpDnLvl.usiValueIdx		:= UDINT_TO_USINT((p_tyUsrMgmtLv3List[udiP1080SelectedRow].eUsrLvl) - 1);

			3:
				tyP1080UsrMgmt.tyEdit.tyStringUsrNm.sValue			:= p_tyUsrMgmtAdminList[udiP1080SelectedRow].sUsrNm;
				tyP1080UsrMgmt.tyEdit.tyDrpDnLvl.usiValueIdx		:= UDINT_TO_USINT((p_tyUsrMgmtAdminList[udiP1080SelectedRow].eUsrLvl) - 1);
		END_CASE

		tyP1080UsrMgmt.tyEdit.tyStringPw.sValue						:= '';

		IF usiP1080SelectedLvl = 5 OR usiP1080SelectedLvl = 6 THEN
			tyP1080UsrMgmt.tyEdit.tyDrpDnLvl.usiValueMinIdx			:= 3;
			tyP1080UsrMgmt.tyEdit.tyDrpDnLvl.usiValueMaxIdx			:= 4;
		ELSE
			tyP1080UsrMgmt.tyEdit.tyDrpDnLvl.usiValueMinIdx			:= 0;
			tyP1080UsrMgmt.tyEdit.tyDrpDnLvl.usiValueMaxIdx			:= 2;
		END_IF

		tyP1080UsrMgmt.tyUsrMgmt.tyBtnEditDetail.bRtCompl			:= FALSE;
		tyP1080UsrMgmt.tyUsrMgmt.tyBtnEditDetail.bValue				:= TRUE;

	END_IF

	// Edit User
	IF tyP1080UsrMgmt.tyUsrMgmt.tyBtnEditDetail.bValue = TRUE THEN
		IF tyP1080UsrMgmt.tyEdit.tyBtnOk.bRtCompl = TRUE THEN
			IF usiEditUsrMgmtStep = 0 THEN
				tyUsrMgmtInfoIn.sUsrNm			:= tyP1080UsrMgmt.tyEdit.tyStringUsrNm.sValue;
				tyUsrMgmtInfoIn.sPw				:= tyP1080UsrMgmt.tyEdit.tyStringPw.sValue;
				tyUsrMgmtInfoIn.eUsrLvl			:= tyP1080UsrMgmt.tyEdit.tyDrpDnLvl.usiValueIdx + 1;

				eUsrMgmtAct					:= UsrMgmtActEdit;

				IF p_eUsrMgmtStat = UsrMgmtActEdit AND p_eUsrMgmtStatus = Done THEN
					eUsrMgmtAct				:= UsrMgmtActIdle;

					IF p_bUsrMgmtNmEmpty = TRUE THEN
						usiEditUsrMgmtStep		:= 1;
					ELSIF p_bUsrMgmtListFull = TRUE THEN
						usiEditUsrMgmtStep		:= 2;
					ELSE
						bRefreshUsrMgmtTable	:= TRUE;
						usiEditUsrMgmtStep		:= 99;
					END_IF
				ELSIF p_eUsrMgmtStatus = Error THEN
					p_tyC0008MsgBox ACCESS ADR(tyP1080UsrMgmt.tyMsgBoxEditErr);

					IF tyP1080UsrMgmt.tyMsgBoxEditErr.tyBtnNo.bRtCompl = TRUE THEN
						tyP1080UsrMgmt.tyMsgBoxEditErr.tyBtnNo.bRtCompl 		:= FALSE;
						tyP1080UsrMgmt.tyMsgBoxEditErr.tyBtnNo.bValue 			:= FALSE;

						p_tyC0008MsgBox ACCESS ADR(tyP1080UsrMgmt.tyMsgBoxHide);

						usiEditUsrMgmtStep		:= 99;
					END_IF
				END_IF

			// User Managment Param Invalid
			ELSIF usiEditUsrMgmtStep = 1 THEN
				p_tyC0008MsgBox ACCESS ADR(tyP1080UsrMgmt.tyMsgBoxEditParamErr);

				IF tyP1080UsrMgmt.tyMsgBoxEditParamErr.tyBtnNo.bRtCompl = TRUE THEN
					tyP1080UsrMgmt.tyMsgBoxEditParamErr.tyBtnNo.bRtCompl 		:= FALSE;
					tyP1080UsrMgmt.tyMsgBoxEditParamErr.tyBtnNo.bValue 			:= FALSE;

					p_tyC0008MsgBox ACCESS ADR(tyP1040ProdSet.tyMsgBoxHide);

					tyP1080UsrMgmt.tyEdit.tyStringPw.sValue						:= '';
					tyP1080UsrMgmt.tyEdit.tyDrpDnLvl.usiValueIdx				:= 0;

					tyP1080UsrMgmt.tyEdit.tyBtnOk.bRtCompl 						:= FALSE;
					tyP1080UsrMgmt.tyEdit.tyBtnOk.bValue 						:= FALSE;

					usiEditUsrMgmtStep			:= 0;
				END_IF

			// User Managment List Full
			ELSIF usiEditUsrMgmtStep = 2 THEN
				p_tyC0008MsgBox ACCESS ADR(tyP1080UsrMgmt.tyMsgBoxListFull);

				IF tyP1080UsrMgmt.tyMsgBoxListFull.tyBtnNo.bRtCompl = TRUE THEN
					tyP1080UsrMgmt.tyMsgBoxListFull.tyBtnNo.bRtCompl 			:= FALSE;
					tyP1080UsrMgmt.tyMsgBoxListFull.tyBtnNo.bValue 				:= FALSE;

					p_tyC0008MsgBox ACCESS ADR(tyP1080UsrMgmt.tyMsgBoxHide);

					usiEditUsrMgmtStep			:= 99;
				END_IF

			ELSIF usiEditUsrMgmtStep = 99 THEN
				fUIInRtStatOff(ADR(tyP1080UsrMgmt.tyUsrMgmt.tyLyr.uiRtStat));
				fUIInRtStatHide(ADR(tyP1080UsrMgmt.tyEdit.tyLyr.uiRtStat));

				tyP1080UsrMgmt.tyUsrMgmt.tyBtnEditDetail.bValue					:= FALSE;

				tyP1080UsrMgmt.tyEdit.tyBtnOk.bRtCompl							:= FALSE;
				tyP1080UsrMgmt.tyEdit.tyBtnOk.bValue							:= FALSE;

				usiEditUsrMgmtStep				:= 0;
			END_IF

		ELSIF tyP1080UsrMgmt.tyEdit.tyBtnCancel.bRtCompl = TRUE THEN
			fUIInRtStatOff(ADR(tyP1080UsrMgmt.tyUsrMgmt.tyLyr.uiRtStat));
			fUIInRtStatHide(ADR(tyP1080UsrMgmt.tyEdit.tyLyr.uiRtStat));

			tyP1080UsrMgmt.tyUsrMgmt.tyBtnEditDetail.bValue						:= FALSE;

			tyP1080UsrMgmt.tyEdit.tyBtnCancel.bRtCompl							:= FALSE;
			tyP1080UsrMgmt.tyEdit.tyBtnCancel.bValue							:= FALSE;
		END_IF
	END_IF

END_ACTION
```

#### Act_OptP1080Keypad.st
```iecst
ACTION Act_OptP1080Keypad:

	IF fUIOutRtStatTPIsOpen(ADR(tyP1080UsrMgmt.tyCreate.tyStringUsrNm.uiRtStat)) = TRUE THEN
		tyProperty.tyKeypad.tyTxtTitle.sTxt	:= tyP1080UsrMgmt.tyCreate.tyStringUsrNm.sKeypadTitle;

	ELSIF fUIOutRtStatTPIsOpen(ADR(tyP1080UsrMgmt.tyCreate.tyStringPw.uiRtStat)) = TRUE THEN
		tyProperty.tyKeypad.tyTxtTitle.sTxt	:= tyP1080UsrMgmt.tyCreate.tyStringPw.sKeypadTitle;

	ELSIF fUIOutRtStatTPIsOpen(ADR(tyP1080UsrMgmt.tyEdit.tyStringPw.uiRtStat)) = TRUE THEN
		tyProperty.tyKeypad.tyTxtTitle.sTxt	:= tyP1080UsrMgmt.tyCreate.tyStringPw.sKeypadTitle;

	END_IF

END_ACTION
```

#### Act_OptP1080Table.st
```iecst
ACTION Act_OptP1080Table:

	fbP1080Table.sVisuNm			:= tyP1080Table.sVisuNm;
	fbP1080Table.udiWorkAreaStartX	:= 50;
	fbP1080Table.udiWorkAreaEndX	:= 497;
	fbP1080Table.udiWorkAreaStartY	:= 109;
	fbP1080Table.udiWorkAreaEndY	:= 458;
	fbP1080Table.udiMinXDist		:= 20;
	fbP1080Table.udiMinYDist		:= 20;
	fbP1080Table.uiSlideScale		:= c_uiP1080TableSize;
	fbP1080Table.iTotalData			:= UDINT_TO_INT(c_udiUsrMgmtMax);
	fbP1080Table.iTotalRow			:= c_uiP1080TableSize;
	fbP1080Table(uiSliderStatus := tyP1080UsrMgmt.tyUsrMgmt.tyTableList.tyUISlider.uiRtStat , a_tyUIHotspot := tyP1080UsrMgmt.tyUsrMgmt.tyTableList.a_tyHotspot , uiTablePos := tyP1080Table.uiTablePos , iSliderPos := tyP1080UsrMgmt.tyUsrMgmt.tyTableList.tyUISlider.iValue);

	tyP1080Table.uiSelectedRow		:= fbP1080Table.uiSelectedRow;
	tyP1080Table.bTableActive		:= fbP1080Table.bTableActive;
	tyP1080Table.bSliderActive		:= fbP1080Table.bSliderActive;

	//Table Content
	IF tyP1080Table.bTableActive = TRUE OR tyP1080Table.bSliderActive = TRUE OR bRefreshUsrMgmtTable = TRUE THEN
		FOR i := 1 TO c_uiP1080TableSize DO

			tyP1080UsrMgmt.tyUsrMgmt.tyTableList.a_tyStringDataCol0[i].sValue				:= UINT_TO_STRING(tyP1080Table.uiTablePos + i - 1);

			CASE tyP1080UsrMgmt.tyUsrMgmt.tyDrpDnLvl.usiValueIdx OF
				// User All
				0:
					tyP1080UsrMgmt.tyUsrMgmt.tyTableList.a_tyStringDataCol1[i].sValue		:= p_tyUsrMgmtAllList[tyP1080Table.uiTablePos + i - 1].sUsrNm;
					tyP1080UsrMgmt.tyUsrMgmt.tyTableList.a_tyTxtDataCol3[i].usiValueIdx		:= DINT_TO_USINT(p_tyUsrMgmtAllList[tyP1080Table.uiTablePos + i - 1].eUsrLvl + 1);
				// User Level 2
				1:
					tyP1080UsrMgmt.tyUsrMgmt.tyTableList.a_tyStringDataCol1[i].sValue		:= p_tyUsrMgmtLv2List[tyP1080Table.uiTablePos + i - 1].sUsrNm;
					tyP1080UsrMgmt.tyUsrMgmt.tyTableList.a_tyTxtDataCol3[i].usiValueIdx		:= DINT_TO_USINT(p_tyUsrMgmtLv2List[tyP1080Table.uiTablePos + i - 1].eUsrLvl + 1);
				// User Level 3
				2:
					tyP1080UsrMgmt.tyUsrMgmt.tyTableList.a_tyStringDataCol1[i].sValue		:= p_tyUsrMgmtLv3List[tyP1080Table.uiTablePos + i - 1].sUsrNm;
					tyP1080UsrMgmt.tyUsrMgmt.tyTableList.a_tyTxtDataCol3[i].usiValueIdx		:= DINT_TO_USINT(p_tyUsrMgmtLv3List[tyP1080Table.uiTablePos + i - 1].eUsrLvl + 1);
				// User Admin
				3:
					tyP1080UsrMgmt.tyUsrMgmt.tyTableList.a_tyStringDataCol1[i].sValue		:= p_tyUsrMgmtAdminList[tyP1080Table.uiTablePos + i - 1].sUsrNm;
					tyP1080UsrMgmt.tyUsrMgmt.tyTableList.a_tyTxtDataCol3[i].usiValueIdx		:= DINT_TO_USINT(p_tyUsrMgmtAdminList[tyP1080Table.uiTablePos + i - 1].eUsrLvl + 1);
			END_CASE
		END_FOR
		bRefreshUsrMgmtTable 			:= FALSE;
	END_IF

	IF tyP1080UsrMgmt.tyUsrMgmt.tyDrpDnLvl.bRtCompl = TRUE THEN
		tyP1080UsrMgmt.tyUsrMgmt.tyDrpDnLvl.bRtCompl	:= FALSE;
		bRefreshUsrMgmtTable 							:= TRUE;
	END_IF

	//Selected Row
	IF tyP1080Table.uiSelectedRow <> tyP1080Table.uiSelectedRowOld THEN
		FOR i := 1 TO c_uiP1080TableSize DO
			IF tyP1080Table.uiSelectedRow = i THEN
				tyP1080UsrMgmt.tyUsrMgmt.tyTableList.a_tyStringDataCol1[i].usiColor		:= 1;
				tyP1080UsrMgmt.tyUsrMgmt.tyTableList.a_tyTxtDataCol3[i].usiColor		:= 1;

			ELSE
				tyP1080UsrMgmt.tyUsrMgmt.tyTableList.a_tyStringDataCol1[i].usiColor		:= 0;
				tyP1080UsrMgmt.tyUsrMgmt.tyTableList.a_tyTxtDataCol3[i].usiColor		:= 0;

			END_IF
		END_FOR

		tyP1080Table.uiSelectedRowOld	:= tyP1080Table.uiSelectedRow;

	END_IF

	IF tyP1080UsrMgmt.tyUsrMgmt.tyTableList.a_tyStringDataCol1[tyP1080Table.uiSelectedRow].sValue = '' THEN
		fUIInRtStatOff(ADR(tyP1080UsrMgmt.tyUsrMgmt.tyBtnEditDetail.uiMaskRtStat));
		fUIInRtStatOff(ADR(tyP1080UsrMgmt.tyUsrMgmt.tyBtnDeleteUsr.uiMaskRtStat));
	ELSE
		fUIInRtStatHide(ADR(tyP1080UsrMgmt.tyUsrMgmt.tyBtnEditDetail.uiMaskRtStat));
		fUIInRtStatHide(ADR(tyP1080UsrMgmt.tyUsrMgmt.tyBtnDeleteUsr.uiMaskRtStat));
	END_IF

END_ACTION
```

#### Act_EntP1081Disp.st
```iecst
ACTION Act_EntP1081Disp:

	//Access Address
	p_tyC0004Navi ACCESS ADR(tyP1081UsrMgmtUsrAccessRgt.tyNaviBack);

	p_tyC0005Main ACCESS ADR(tyCommon.tyMain);

	p_tyC0006Set ACCESS ADR(tyCommon.tySet);

	p_tyC0007Notif ACCESS ADR(tyCommon.tyNotif);

	p_tyC0008MsgBox ACCESS ADR(tyP1081UsrMgmtUsrAccessRgt.tyMsgBoxHide);

	p_tyC0009Info ACCESS ADR(tyCommon.tyInfo);

	p_tyC0011Loading ACCESS ADR(tyCommon.tyLoading);

	p_tyP1081UsrMgmtUsrAccessRgtSel ACCESS ADR(tyP1081UsrMgmtUsrAccessRgt.tyUsrAccessRgtSel);
	p_tyP1081UsrMgmtUsrAccessRgt ACCESS ADR(tyP1081UsrMgmtUsrAccessRgt.tyUsrAccessRgtLvl1);

	//Display
	//Reset DrpDn List
	tyP1081UsrMgmtUsrAccessRgt.tyUsrAccessRgtSel.tyDrpDnLevel.usiValueIdx	:= 0;

	//Backup Param
	tyP1081UsrMgmtUsrAccessRgt.tyUsrAccessRgtLvl1BkUp	:= tyP1081UsrMgmtUsrAccessRgt.tyUsrAccessRgtLvl1;
	tyP1081UsrMgmtUsrAccessRgt.tyUsrAccessRgtLvl2BkUp	:= tyP1081UsrMgmtUsrAccessRgt.tyUsrAccessRgtLvl2;
	tyP1081UsrMgmtUsrAccessRgt.tyUsrAccessRgtLvl3BkUp	:= tyP1081UsrMgmtUsrAccessRgt.tyUsrAccessRgtLvl3;

END_ACTION
```

#### Act_ExitP1081.st
```iecst
ACTION Act_ExitP1081:

	IF tyCommon.tySet.tyBtnSave.uiMaskRtStat.0 = FALSE THEN
		usiChgPage	:= 1;

	ELSE

		p_tyC0008MsgBox ACCESS ADR(tyP1081UsrMgmtUsrAccessRgt.tyMsgBoxExitAsk);

		IF tyP1081UsrMgmtUsrAccessRgt.tyMsgBoxExitAsk.tyBtnYes.bRtCompl = TRUE THEN
			tyP1081UsrMgmtUsrAccessRgt.tyMsgBoxExitAsk.tyBtnYes.bRtCompl	:= FALSE;
			tyP1081UsrMgmtUsrAccessRgt.tyMsgBoxExitAsk.tyBtnYes.bValue		:= FALSE;

			p_tyC0008MsgBox ACCESS ADR(tyP1081UsrMgmtUsrAccessRgt.tyMsgBoxHide);

			//Restore Param
			tyP1081UsrMgmtUsrAccessRgt.tyUsrAccessRgtLvl1	:= tyP1081UsrMgmtUsrAccessRgt.tyUsrAccessRgtLvl1BkUp;
			tyP1081UsrMgmtUsrAccessRgt.tyUsrAccessRgtLvl2	:= tyP1081UsrMgmtUsrAccessRgt.tyUsrAccessRgtLvl2BkUp;
			tyP1081UsrMgmtUsrAccessRgt.tyUsrAccessRgtLvl3	:= tyP1081UsrMgmtUsrAccessRgt.tyUsrAccessRgtLvl3BkUp;

			fUIInRtStatOff(ADR(tyCommon.tySet.tyBtnSave.uiMaskRtStat));

			usiChgPage	:= 1;

		ELSIF tyP1081UsrMgmtUsrAccessRgt.tyMsgBoxExitAsk.tyBtnNo.bRtCompl = TRUE THEN
			tyP1081UsrMgmtUsrAccessRgt.tyMsgBoxExitAsk.tyBtnNo.bRtCompl	:= FALSE;
			tyP1081UsrMgmtUsrAccessRgt.tyMsgBoxExitAsk.tyBtnNo.bValue	:= FALSE;

			p_tyC0008MsgBox ACCESS ADR(tyP1081UsrMgmtUsrAccessRgt.tyMsgBoxHide);

			eChgPage	:= eCurrPage;
			usiChgPage	:= 0;

		END_IF

	END_IF

END_ACTION
```
